   1:  PR[GP1:91,1] = PR[GP1:90,1] + -48.523;
   1:  PR[GP1:91,2] = PR[GP1:90,2] + 33.030;
   1:L PR[91] R[100]mm/sec CNT100;
   1:  PR[GP1:91,1] = PR[GP1:90,1] + -49.948;
   1:  PR[GP1:91,2] = PR[GP1:90,2] + 32.411;
   1:L PR[91] R[100]mm/sec CNT100;
   1:  PR[GP1:91,1] = PR[GP1:90,1] + -58.284;
   1:  PR[GP1:91,2] = PR[GP1:90,2] + 28.248;
   1:L PR[91] R[100]mm/sec CNT100;
   1:  PR[GP1:91,1] = PR[GP1:90,1] + -60.456;
   1:  PR[GP1:91,2] = PR[GP1:90,2] + 26.266;
   1:L PR[91] R[100]mm/sec CNT100;
   1:  PR[GP1:91,1] = PR[GP1:90,1] + -66.187;
   1:  PR[GP1:91,2] = PR[GP1:90,2] + 20.627;
   1:L PR[91] R[100]mm/sec CNT100;
   1:  PR[GP1:91,1] = PR[GP1:90,1] + -68.044;
   1:  PR[GP1:91,2] = PR[GP1:90,2] + 17.225;
   1:L PR[91] R[100]mm/sec CNT100;
   1:  PR[GP1:91,1] = PR[GP1:90,1] + -71.335;
   1:  PR[GP1:91,2] = PR[GP1:90,2] + 10.856;
   1:L PR[91] R[100]mm/sec CNT100;
   1:  PR[GP1:91,1] = PR[GP1:90,1] + -72.085;
   1:  PR[GP1:91,2] = PR[GP1:90,2] + 6.431;
   1:L PR[91] R[100]mm/sec CNT100;
   1:  PR[GP1:91,1] = PR[GP1:90,1] + -73.126;
   1:  PR[GP1:91,2] = PR[GP1:90,2] + -0.069;
   1:L PR[91] R[100]mm/sec CNT100;
   1:  PR[GP1:91,1] = PR[GP1:90,1] + -72.374;
   1:  PR[GP1:91,2] = PR[GP1:90,2] + -4.503;
   1:L PR[91] R[100]mm/sec CNT100;
   1:  PR[GP1:91,1] = PR[GP1:90,1] + -71.334;
   1:  PR[GP1:91,2] = PR[GP1:90,2] + -11.003;
   1:L PR[91] R[100]mm/sec CNT100;
   1:  PR[GP1:91,1] = PR[GP1:90,1] + -68.044;
   1:  PR[GP1:91,2] = PR[GP1:90,2] + -17.369;
   1:L PR[91] R[100]mm/sec CNT100;
   1:  PR[GP1:91,1] = PR[GP1:90,1] + -66.187;
   1:  PR[GP1:91,2] = PR[GP1:90,2] + -20.771;
   1:L PR[91] R[100]mm/sec CNT100;
   1:  PR[GP1:91,1] = PR[GP1:90,1] + -60.456;
   1:  PR[GP1:91,2] = PR[GP1:90,2] + -26.411;
   1:L PR[91] R[100]mm/sec CNT100;
   1:  PR[GP1:91,1] = PR[GP1:90,1] + -58.284;
   1:  PR[GP1:91,2] = PR[GP1:90,2] + -28.392;
   1:L PR[91] R[100]mm/sec CNT100;
   1:  PR[GP1:91,1] = PR[GP1:90,1] + -49.948;
   1:  PR[GP1:91,2] = PR[GP1:90,2] + -32.555;
   1:L PR[91] R[100]mm/sec CNT100;
   1:  PR[GP1:91,1] = PR[GP1:90,1] + -48.524;
   1:  PR[GP1:91,2] = PR[GP1:90,2] + -33.174;
   1:L PR[91] R[100]mm/sec CNT100;
   1:  PR[GP1:91,1] = PR[GP1:90,1] + -37.881;
   1:  PR[GP1:91,2] = PR[GP1:90,2] + -34.799;
   1:L PR[91] R[100]mm/sec CNT100;
   1:  PR[GP1:91,1] = PR[GP1:90,1] + -37.801;
   1:  PR[GP1:91,2] = PR[GP1:90,2] + -34.793;
   1:L PR[91] R[100]mm/sec CNT100;
   1:  PR[GP1:91,1] = PR[GP1:90,1] + -27.317;
   1:  PR[GP1:91,2] = PR[GP1:90,2] + -33.256;
   1:L PR[91] R[100]mm/sec CNT100;
   1:  PR[GP1:91,1] = PR[GP1:90,1] + -25.233;
   1:  PR[GP1:91,2] = PR[GP1:90,2] + -32.463;
   1:L PR[91] R[100]mm/sec CNT100;
   1:  PR[GP1:91,1] = PR[GP1:90,1] + -17.847;
   1:  PR[GP1:91,2] = PR[GP1:90,2] + -28.861;
   1:L PR[91] R[100]mm/sec CNT100;
   1:  PR[GP1:91,1] = PR[GP1:90,1] + -14.429;
   1:  PR[GP1:91,2] = PR[GP1:90,2] + -26.222;
   1:L PR[91] R[100]mm/sec CNT100;
   1:  PR[GP1:91,1] = PR[GP1:90,1] + -10.165;
   1:  PR[GP1:91,2] = PR[GP1:90,2] + -22.104;
   1:L PR[91] R[100]mm/sec CNT100;
   1:  PR[GP1:91,1] = PR[GP1:90,1] + -6.579;
   1:  PR[GP1:91,2] = PR[GP1:90,2] + -16.904;
   1:L PR[91] R[100]mm/sec CNT100;
   1:  PR[GP1:91,1] = PR[GP1:90,1] + -4.548;
   1:  PR[GP1:91,2] = PR[GP1:90,2] + -13.017;
   1:L PR[91] R[100]mm/sec CNT100;
   1:  PR[GP1:91,1] = PR[GP1:90,1] + -4.423;
   1:  PR[GP1:91,2] = PR[GP1:90,2] + -13.058;
   1:L PR[91] R[100]mm/sec CNT100;
   1:  PR[GP1:91,1] = PR[GP1:90,1] + -2.556;
   1:  PR[GP1:91,2] = PR[GP1:90,2] + -11.014;
   1:L PR[91] R[100]mm/sec CNT100;
   1:  PR[GP1:91,1] = PR[GP1:90,1] + -1.961;
   1:  PR[GP1:91,2] = PR[GP1:90,2] + -10.303;
   1:L PR[91] R[100]mm/sec CNT100;
   1:  PR[GP1:91,1] = PR[GP1:90,1] + -1.561;
   1:  PR[GP1:91,2] = PR[GP1:90,2] + -10.351;
   1:L PR[91] R[100]mm/sec CNT100;
   1:  PR[GP1:91,1] = PR[GP1:90,1] + 2.228;
   1:  PR[GP1:91,2] = PR[GP1:90,2] + -10.312;
   1:L PR[91] R[100]mm/sec CNT100;
   1:  PR[GP1:91,1] = PR[GP1:90,1] + 2.419;
   1:  PR[GP1:91,2] = PR[GP1:90,2] + -10.673;
   1:L PR[91] R[100]mm/sec CNT100;
   1:  PR[GP1:91,1] = PR[GP1:90,1] + 2.721;
   1:  PR[GP1:91,2] = PR[GP1:90,2] + -11.007;
   1:L PR[91] R[100]mm/sec CNT100;
   1:  PR[GP1:91,1] = PR[GP1:90,1] + 4.385;
   1:  PR[GP1:91,2] = PR[GP1:90,2] + -12.999;
   1:L PR[91] R[100]mm/sec CNT100;
   1:  PR[GP1:91,1] = PR[GP1:90,1] + 4.919;
   1:  PR[GP1:91,2] = PR[GP1:90,2] + -13.336;
   1:L PR[91] R[100]mm/sec CNT100;
   1:  PR[GP1:91,1] = PR[GP1:90,1] + 6.783;
   1:  PR[GP1:91,2] = PR[GP1:90,2] + -16.884;
   1:L PR[91] R[100]mm/sec CNT100;
   1:  PR[GP1:91,1] = PR[GP1:90,1] + 10.374;
   1:  PR[GP1:91,2] = PR[GP1:90,2] + -22.091;
   1:L PR[91] R[100]mm/sec CNT100;
   1:  PR[GP1:91,1] = PR[GP1:90,1] + 14.635;
   1:  PR[GP1:91,2] = PR[GP1:90,2] + -26.217;
   1:L PR[91] R[100]mm/sec CNT100;
   1:  PR[GP1:91,1] = PR[GP1:90,1] + 18.052;
   1:  PR[GP1:91,2] = PR[GP1:90,2] + -28.858;
   1:L PR[91] R[100]mm/sec CNT100;
   1:  PR[GP1:91,1] = PR[GP1:90,1] + 25.434;
   1:  PR[GP1:91,2] = PR[GP1:90,2] + -32.459;
   1:L PR[91] R[100]mm/sec CNT100;
   1:  PR[GP1:91,1] = PR[GP1:90,1] + 27.520;
   1:  PR[GP1:91,2] = PR[GP1:90,2] + -33.250;
   1:L PR[91] R[100]mm/sec CNT100;
   1:  PR[GP1:91,1] = PR[GP1:90,1] + 38.001;
   1:  PR[GP1:91,2] = PR[GP1:90,2] + -34.793;
   1:L PR[91] R[100]mm/sec CNT100;
   1:  PR[GP1:91,1] = PR[GP1:90,1] + 38.083;
   1:  PR[GP1:91,2] = PR[GP1:90,2] + -34.799;
   1:L PR[91] R[100]mm/sec CNT100;
   1:  PR[GP1:91,1] = PR[GP1:90,1] + 48.729;
   1:  PR[GP1:91,2] = PR[GP1:90,2] + -33.175;
   1:L PR[91] R[100]mm/sec CNT100;
   1:  PR[GP1:91,1] = PR[GP1:90,1] + 50.153;
   1:  PR[GP1:91,2] = PR[GP1:90,2] + -32.556;
   1:L PR[91] R[100]mm/sec CNT100;
   1:  PR[GP1:91,1] = PR[GP1:90,1] + 58.492;
   1:  PR[GP1:91,2] = PR[GP1:90,2] + -28.398;
   1:L PR[91] R[100]mm/sec CNT100;
   1:  PR[GP1:91,1] = PR[GP1:90,1] + 60.665;
   1:  PR[GP1:91,2] = PR[GP1:90,2] + -26.416;
   1:L PR[91] R[100]mm/sec CNT100;
   1:  PR[GP1:91,1] = PR[GP1:90,1] + 66.398;
   1:  PR[GP1:91,2] = PR[GP1:90,2] + -20.767;
   1:L PR[91] R[100]mm/sec CNT100;
   1:  PR[GP1:91,1] = PR[GP1:90,1] + 68.256;
   1:  PR[GP1:91,2] = PR[GP1:90,2] + -17.367;
   1:L PR[91] R[100]mm/sec CNT100;
   1:  PR[GP1:91,1] = PR[GP1:90,1] + 71.548;
   1:  PR[GP1:91,2] = PR[GP1:90,2] + -11.013;
   1:L PR[91] R[100]mm/sec CNT100;
   1:  PR[GP1:91,1] = PR[GP1:90,1] + 72.297;
   1:  PR[GP1:91,2] = PR[GP1:90,2] + -6.586;
   1:L PR[91] R[100]mm/sec CNT100;
   1:  PR[GP1:91,1] = PR[GP1:90,1] + 73.340;
   1:  PR[GP1:91,2] = PR[GP1:90,2] + -0.075;
   1:L PR[91] R[100]mm/sec CNT100;
   1:  PR[GP1:91,1] = PR[GP1:90,1] + 72.588;
   1:  PR[GP1:91,2] = PR[GP1:90,2] + 4.361;
   1:L PR[91] R[100]mm/sec CNT100;
   1:  PR[GP1:91,1] = PR[GP1:90,1] + 71.547;
   1:  PR[GP1:91,2] = PR[GP1:90,2] + 10.872;
   1:L PR[91] R[100]mm/sec CNT100;
   1:  PR[GP1:91,1] = PR[GP1:90,1] + 68.256;
   1:  PR[GP1:91,2] = PR[GP1:90,2] + 17.223;
   1:L PR[91] R[100]mm/sec CNT100;
   1:  PR[GP1:91,1] = PR[GP1:90,1] + 66.398;
   1:  PR[GP1:91,2] = PR[GP1:90,2] + 20.623;
   1:L PR[91] R[100]mm/sec CNT100;
   1:  PR[GP1:91,1] = PR[GP1:90,1] + 60.665;
   1:  PR[GP1:91,2] = PR[GP1:90,2] + 26.272;
   1:L PR[91] R[100]mm/sec CNT100;
   1:  PR[GP1:91,1] = PR[GP1:90,1] + 58.492;
   1:  PR[GP1:91,2] = PR[GP1:90,2] + 28.254;
   1:L PR[91] R[100]mm/sec CNT100;
   1:  PR[GP1:91,1] = PR[GP1:90,1] + 50.152;
   1:  PR[GP1:91,2] = PR[GP1:90,2] + 32.412;
   1:L PR[91] R[100]mm/sec CNT100;
   1:  PR[GP1:91,1] = PR[GP1:90,1] + 48.729;
   1:  PR[GP1:91,2] = PR[GP1:90,2] + 33.031;
   1:L PR[91] R[100]mm/sec CNT100;
   1:  PR[GP1:91,1] = PR[GP1:90,1] + 38.083;
   1:  PR[GP1:91,2] = PR[GP1:90,2] + 34.655;
   1:L PR[91] R[100]mm/sec CNT100;
   1:  PR[GP1:91,1] = PR[GP1:90,1] + 38.001;
   1:  PR[GP1:91,2] = PR[GP1:90,2] + 34.649;
   1:L PR[91] R[100]mm/sec CNT100;
   1:  PR[GP1:91,1] = PR[GP1:90,1] + 27.520;
   1:  PR[GP1:91,2] = PR[GP1:90,2] + 33.106;
   1:L PR[91] R[100]mm/sec CNT100;
   1:  PR[GP1:91,1] = PR[GP1:90,1] + 25.434;
   1:  PR[GP1:91,2] = PR[GP1:90,2] + 32.314;
   1:L PR[91] R[100]mm/sec CNT100;
   1:  PR[GP1:91,1] = PR[GP1:90,1] + 18.052;
   1:  PR[GP1:91,2] = PR[GP1:90,2] + 28.714;
   1:L PR[91] R[100]mm/sec CNT100;
   1:  PR[GP1:91,1] = PR[GP1:90,1] + 14.635;
   1:  PR[GP1:91,2] = PR[GP1:90,2] + 26.073;
   1:L PR[91] R[100]mm/sec CNT100;
   1:  PR[GP1:91,1] = PR[GP1:90,1] + 10.374;
   1:  PR[GP1:91,2] = PR[GP1:90,2] + 21.947;
   1:L PR[91] R[100]mm/sec CNT100;
   1:  PR[GP1:91,1] = PR[GP1:90,1] + 6.797;
   1:  PR[GP1:91,2] = PR[GP1:90,2] + 16.767;
   1:L PR[91] R[100]mm/sec CNT100;
   1:  PR[GP1:91,1] = PR[GP1:90,1] + 4.956;
   1:  PR[GP1:91,2] = PR[GP1:90,2] + 13.264;
   1:L PR[91] R[100]mm/sec CNT100;
   1:  PR[GP1:91,1] = PR[GP1:90,1] + 2.737;
   1:  PR[GP1:91,2] = PR[GP1:90,2] + 10.879;
   1:L PR[91] R[100]mm/sec CNT100;
   1:  PR[GP1:91,1] = PR[GP1:90,1] + 2.140;
   1:  PR[GP1:91,2] = PR[GP1:90,2] + 10.164;
   1:L PR[91] R[100]mm/sec CNT100;
   1:  PR[GP1:91,1] = PR[GP1:90,1] + -1.651;
   1:  PR[GP1:91,2] = PR[GP1:90,2] + 10.194;
   1:L PR[91] R[100]mm/sec CNT100;
   1:  ! -- Layer/Ebene 45 -- !;
   1:  PR[91] = PR[90];
   1:  PR[GP1:91,1] = PR[GP1:90,1] + -2.160;
   1:  PR[GP1:91,2] = PR[GP1:90,2] + 10.865;
   1:  PR[GP1:91,3] = PR[GP1:90,3] + 27.755;
   1:L PR[91] R[100]mm/sec CNT100;
   1:  PR[GP1:91,1] = PR[GP1:90,1] + -4.791;
   1:  PR[GP1:91,2] = PR[GP1:90,2] + 13.704;
   1:L PR[91] R[100]mm/sec CNT100;
   1:  PR[GP1:91,1] = PR[GP1:90,1] + -4.807;
   1:  PR[GP1:91,2] = PR[GP1:90,2] + 13.843;
   1:L PR[91] R[100]mm/sec CNT100;
   1:  PR[GP1:91,1] = PR[GP1:90,1] + -6.082;
   1:  PR[GP1:91,2] = PR[GP1:90,2] + 16.274;
   1:L PR[91] R[100]mm/sec CNT100;
   1:  PR[GP1:91,1] = PR[GP1:90,1] + -10.209;
   1:  PR[GP1:91,2] = PR[GP1:90,2] + 22.252;
   1:L PR[91] R[100]mm/sec CNT100;
   1:  PR[GP1:91,1] = PR[GP1:90,1] + -13.777;
   1:  PR[GP1:91,2] = PR[GP1:90,2] + 25.698;
   1:L PR[91] R[100]mm/sec CNT100;
   1:  PR[GP1:91,1] = PR[GP1:90,1] + -17.920;
   1:  PR[GP1:91,2] = PR[GP1:90,2] + 28.896;
   1:L PR[91] R[100]mm/sec CNT100;
   1:  PR[GP1:91,1] = PR[GP1:90,1] + -24.472;
   1:  PR[GP1:91,2] = PR[GP1:90,2] + 32.093;
   1:L PR[91] R[100]mm/sec CNT100;
   1:  PR[GP1:91,1] = PR[GP1:90,1] + -27.383;
   1:  PR[GP1:91,2] = PR[GP1:90,2] + 33.199;
   1:L PR[91] R[100]mm/sec CNT100;
   1:  PR[GP1:91,1] = PR[GP1:90,1] + -37.001;
   1:  PR[GP1:91,2] = PR[GP1:90,2] + 34.610;
   1:L PR[91] R[100]mm/sec CNT100;
   1:  PR[GP1:91,1] = PR[GP1:90,1] + -37.913;
   1:  PR[GP1:91,2] = PR[GP1:90,2] + 34.674;
   1:L PR[91] R[100]mm/sec CNT100;
   1:  PR[GP1:91,1] = PR[GP1:90,1] + -43.210;
   1:  PR[GP1:91,2] = PR[GP1:90,2] + 33.821;
   1:L PR[91] R[100]mm/sec CNT100;
   1:  PR[GP1:91,1] = PR[GP1:90,1] + -48.579;
   1:  PR[GP1:91,2] = PR[GP1:90,2] + 33.005;
   1:L PR[91] R[100]mm/sec CNT100;
   1:  PR[GP1:91,1] = PR[GP1:90,1] + -49.324;
   1:  PR[GP1:91,2] = PR[GP1:90,2] + 32.681;
   1:L PR[91] R[100]mm/sec CNT100;
   1:  PR[GP1:91,1] = PR[GP1:90,1] + -58.292;
   1:  PR[GP1:91,2] = PR[GP1:90,2] + 28.203;
   1:L PR[91] R[100]mm/sec CNT100;
   1:  PR[GP1:91,1] = PR[GP1:90,1] + -59.957;
   1:  PR[GP1:91,2] = PR[GP1:90,2] + 26.684;
   1:L PR[91] R[100]mm/sec CNT100;
   1:  PR[GP1:91,1] = PR[GP1:90,1] + -66.156;
   1:  PR[GP1:91,2] = PR[GP1:90,2] + 20.584;
   1:L PR[91] R[100]mm/sec CNT100;
   1:  PR[GP1:91,1] = PR[GP1:90,1] + -67.704;
   1:  PR[GP1:91,2] = PR[GP1:90,2] + 17.748;
   1:L PR[91] R[100]mm/sec CNT100;
   1:  PR[GP1:91,1] = PR[GP1:90,1] + -71.279;
   1:  PR[GP1:91,2] = PR[GP1:90,2] + 10.831;
   1:L PR[91] R[100]mm/sec CNT100;
   1:  PR[GP1:91,1] = PR[GP1:90,1] + -71.922;
   1:  PR[GP1:91,2] = PR[GP1:90,2] + 7.028;
   1:L PR[91] R[100]mm/sec CNT100;
   1:  PR[GP1:91,1] = PR[GP1:90,1] + -73.060;
   1:  PR[GP1:91,2] = PR[GP1:90,2] + -0.069;
   1:L PR[91] R[100]mm/sec CNT100;
   1:  PR[GP1:91,1] = PR[GP1:90,1] + -72.407;
   1:  PR[GP1:91,2] = PR[GP1:90,2] + -3.918;
   1:L PR[91] R[100]mm/sec CNT100;
   1:  PR[GP1:91,1] = PR[GP1:90,1] + -71.277;
   1:  PR[GP1:91,2] = PR[GP1:90,2] + -10.977;
   1:L PR[91] R[100]mm/sec CNT100;
   1:  PR[GP1:91,1] = PR[GP1:90,1] + -67.704;
   1:  PR[GP1:91,2] = PR[GP1:90,2] + -17.892;
   1:L PR[91] R[100]mm/sec CNT100;
   1:  PR[GP1:91,1] = PR[GP1:90,1] + -66.156;
   1:  PR[GP1:91,2] = PR[GP1:90,2] + -20.728;
   1:L PR[91] R[100]mm/sec CNT100;
   1:  PR[GP1:91,1] = PR[GP1:90,1] + -59.957;
   1:  PR[GP1:91,2] = PR[GP1:90,2] + -26.828;
   1:L PR[91] R[100]mm/sec CNT100;
   1:  PR[GP1:91,1] = PR[GP1:90,1] + -58.292;
   1:  PR[GP1:91,2] = PR[GP1:90,2] + -28.347;
   1:L PR[91] R[100]mm/sec CNT100;
   1:  PR[GP1:91,1] = PR[GP1:90,1] + -49.325;
   1:  PR[GP1:91,2] = PR[GP1:90,2] + -32.825;
   1:L PR[91] R[100]mm/sec CNT100;
   1:  PR[GP1:91,1] = PR[GP1:90,1] + -48.579;
   1:  PR[GP1:91,2] = PR[GP1:90,2] + -33.149;
   1:L PR[91] R[100]mm/sec CNT100;
   1:  PR[GP1:91,1] = PR[GP1:90,1] + -43.210;
   1:  PR[GP1:91,2] = PR[GP1:90,2] + -33.965;
   1:L PR[91] R[100]mm/sec CNT100;
   1:  PR[GP1:91,1] = PR[GP1:90,1] + -37.913;
   1:  PR[GP1:91,2] = PR[GP1:90,2] + -34.818;
   1:L PR[91] R[100]mm/sec CNT100;
   1:  PR[GP1:91,1] = PR[GP1:90,1] + -37.002;
   1:  PR[GP1:91,2] = PR[GP1:90,2] + -34.754;
   1:L PR[91] R[100]mm/sec CNT100;
   1:  PR[GP1:91,1] = PR[GP1:90,1] + -27.383;
   1:  PR[GP1:91,2] = PR[GP1:90,2] + -33.343;
   1:L PR[91] R[100]mm/sec CNT100;
   1:  PR[GP1:91,1] = PR[GP1:90,1] + -24.472;
   1:  PR[GP1:91,2] = PR[GP1:90,2] + -32.237;
   1:L PR[91] R[100]mm/sec CNT100;
   1:  PR[GP1:91,1] = PR[GP1:90,1] + -17.920;
   1:  PR[GP1:91,2] = PR[GP1:90,2] + -29.041;
   1:L PR[91] R[100]mm/sec CNT100;
   1:  PR[GP1:91,1] = PR[GP1:90,1] + -13.777;
   1:  PR[GP1:91,2] = PR[GP1:90,2] + -25.842;
   1:L PR[91] R[100]mm/sec CNT100;
   1:  PR[GP1:91,1] = PR[GP1:90,1] + -10.210;
   1:  PR[GP1:91,2] = PR[GP1:90,2] + -22.396;
   1:L PR[91] R[100]mm/sec CNT100;
   1:  PR[GP1:91,1] = PR[GP1:90,1] + -6.066;
   1:  PR[GP1:91,2] = PR[GP1:90,2] + -16.388;
   1:L PR[91] R[100]mm/sec CNT100;
   1:  PR[GP1:91,1] = PR[GP1:90,1] + -4.516;
   1:  PR[GP1:91,2] = PR[GP1:90,2] + -13.422;
   1:L PR[91] R[100]mm/sec CNT100;
   1:  PR[GP1:91,1] = PR[GP1:90,1] + -4.394;
   1:  PR[GP1:91,2] = PR[GP1:90,2] + -13.462;
   1:L PR[91] R[100]mm/sec CNT100;
   1:  PR[GP1:91,1] = PR[GP1:90,1] + -2.162;
   1:  PR[GP1:91,2] = PR[GP1:90,2] + -11.011;
   1:L PR[91] R[100]mm/sec CNT100;
   1:  PR[GP1:91,1] = PR[GP1:90,1] + -1.823;
   1:  PR[GP1:91,2] = PR[GP1:90,2] + -10.812;
   1:L PR[91] R[100]mm/sec CNT100;
   1:  PR[GP1:91,1] = PR[GP1:90,1] + 2.075;
   1:  PR[GP1:91,2] = PR[GP1:90,2] + -10.774;
   1:L PR[91] R[100]mm/sec CNT100;
   1:  PR[GP1:91,1] = PR[GP1:90,1] + 4.171;
   1:  PR[GP1:91,2] = PR[GP1:90,2] + -13.284;
   1:L PR[91] R[100]mm/sec CNT100;
   1:  PR[GP1:91,1] = PR[GP1:90,1] + 4.886;
   1:  PR[GP1:91,2] = PR[GP1:90,2] + -13.736;
   1:L PR[91] R[100]mm/sec CNT100;
   1:  PR[GP1:91,1] = PR[GP1:90,1] + 6.270;
   1:  PR[GP1:91,2] = PR[GP1:90,2] + -16.369;
   1:L PR[91] R[100]mm/sec CNT100;
   1:  PR[GP1:91,1] = PR[GP1:90,1] + 10.419;
   1:  PR[GP1:91,2] = PR[GP1:90,2] + -22.385;
   1:L PR[91] R[100]mm/sec CNT100;
   1:  PR[GP1:91,1] = PR[GP1:90,1] + 13.984;
   1:  PR[GP1:91,2] = PR[GP1:90,2] + -25.837;
   1:L PR[91] R[100]mm/sec CNT100;
   1:  PR[GP1:91,1] = PR[GP1:90,1] + 18.126;
   1:  PR[GP1:91,2] = PR[GP1:90,2] + -29.039;
   1:L PR[91] R[100]mm/sec CNT100;
   1:  PR[GP1:91,1] = PR[GP1:90,1] + 24.675;
   1:  PR[GP1:91,2] = PR[GP1:90,2] + -32.233;
   1:L PR[91] R[100]mm/sec CNT100;
   1:  PR[GP1:91,1] = PR[GP1:90,1] + 27.587;
   1:  PR[GP1:91,2] = PR[GP1:90,2] + -33.338;
   1:L PR[91] R[100]mm/sec CNT100;
   1:  PR[GP1:91,1] = PR[GP1:90,1] + 37.203;
   1:  PR[GP1:91,2] = PR[GP1:90,2] + -34.754;
   1:L PR[91] R[100]mm/sec CNT100;
   1:  PR[GP1:91,1] = PR[GP1:90,1] + 38.116;
   1:  PR[GP1:91,2] = PR[GP1:90,2] + -34.819;
   1:L PR[91] R[100]mm/sec CNT100;
   1:  PR[GP1:91,1] = PR[GP1:90,1] + 43.423;
   1:  PR[GP1:91,2] = PR[GP1:90,2] + -33.964;
   1:L PR[91] R[100]mm/sec CNT100;
   1:  PR[GP1:91,1] = PR[GP1:90,1] + 48.784;
   1:  PR[GP1:91,2] = PR[GP1:90,2] + -33.150;
   1:L PR[91] R[100]mm/sec CNT100;
   1:  PR[GP1:91,1] = PR[GP1:90,1] + 49.528;
   1:  PR[GP1:91,2] = PR[GP1:90,2] + -32.826;
   1:L PR[91] R[100]mm/sec CNT100;
   1:  PR[GP1:91,1] = PR[GP1:90,1] + 58.500;
   1:  PR[GP1:91,2] = PR[GP1:90,2] + -28.353;
   1:L PR[91] R[100]mm/sec CNT100;
   1:  PR[GP1:91,1] = PR[GP1:90,1] + 60.165;
   1:  PR[GP1:91,2] = PR[GP1:90,2] + -26.835;
   1:L PR[91] R[100]mm/sec CNT100;
   1:  PR[GP1:91,1] = PR[GP1:90,1] + 66.367;
   1:  PR[GP1:91,2] = PR[GP1:90,2] + -20.723;
   1:L PR[91] R[100]mm/sec CNT100;
   1:  PR[GP1:91,1] = PR[GP1:90,1] + 67.915;
   1:  PR[GP1:91,2] = PR[GP1:90,2] + -17.889;
   1:L PR[91] R[100]mm/sec CNT100;
   1:  PR[GP1:91,1] = PR[GP1:90,1] + 71.491;
   1:  PR[GP1:91,2] = PR[GP1:90,2] + -10.988;
   1:L PR[91] R[100]mm/sec CNT100;
   1:  PR[GP1:91,1] = PR[GP1:90,1] + 72.135;
   1:  PR[GP1:91,2] = PR[GP1:90,2] + -7.183;
   1:L PR[91] R[100]mm/sec CNT100;
   1:  PR[GP1:91,1] = PR[GP1:90,1] + 73.273;
   1:  PR[GP1:91,2] = PR[GP1:90,2] + -0.075;
   1:L PR[91] R[100]mm/sec CNT100;
   1:  PR[GP1:91,1] = PR[GP1:90,1] + 72.620;
   1:  PR[GP1:91,2] = PR[GP1:90,2] + 3.775;
   1:L PR[91] R[100]mm/sec CNT100;
   1:  PR[GP1:91,1] = PR[GP1:90,1] + 71.490;
   1:  PR[GP1:91,2] = PR[GP1:90,2] + 10.847;
   1:L PR[91] R[100]mm/sec CNT100;
   1:  PR[GP1:91,1] = PR[GP1:90,1] + 67.915;
   1:  PR[GP1:91,2] = PR[GP1:90,2] + 17.745;
   1:L PR[91] R[100]mm/sec CNT100;
   1:  PR[GP1:91,1] = PR[GP1:90,1] + 66.367;
   1:  PR[GP1:91,2] = PR[GP1:90,2] + 20.579;
   1:L PR[91] R[100]mm/sec CNT100;
   1:  PR[GP1:91,1] = PR[GP1:90,1] + 60.165;
   1:  PR[GP1:91,2] = PR[GP1:90,2] + 26.691;
   1:L PR[91] R[100]mm/sec CNT100;
   1:  PR[GP1:91,1] = PR[GP1:90,1] + 58.500;
   1:  PR[GP1:91,2] = PR[GP1:90,2] + 28.209;
   1:L PR[91] R[100]mm/sec CNT100;
   1:  PR[GP1:91,1] = PR[GP1:90,1] + 49.528;
   1:  PR[GP1:91,2] = PR[GP1:90,2] + 32.682;
   1:L PR[91] R[100]mm/sec CNT100;
   1:  PR[GP1:91,1] = PR[GP1:90,1] + 48.784;
   1:  PR[GP1:91,2] = PR[GP1:90,2] + 33.006;
   1:L PR[91] R[100]mm/sec CNT100;
   1:  PR[GP1:91,1] = PR[GP1:90,1] + 43.423;
   1:  PR[GP1:91,2] = PR[GP1:90,2] + 33.820;
   1:L PR[91] R[100]mm/sec CNT100;
   1:  PR[GP1:91,1] = PR[GP1:90,1] + 38.116;
   1:  PR[GP1:91,2] = PR[GP1:90,2] + 34.675;
   1:L PR[91] R[100]mm/sec CNT100;
   1:  PR[GP1:91,1] = PR[GP1:90,1] + 37.203;
   1:  PR[GP1:91,2] = PR[GP1:90,2] + 34.610;
   1:L PR[91] R[100]mm/sec CNT100;
   1:  PR[GP1:91,1] = PR[GP1:90,1] + 27.586;
   1:  PR[GP1:91,2] = PR[GP1:90,2] + 33.194;
   1:L PR[91] R[100]mm/sec CNT100;
   1:  PR[GP1:91,1] = PR[GP1:90,1] + 24.675;
   1:  PR[GP1:91,2] = PR[GP1:90,2] + 32.089;
   1:L PR[91] R[100]mm/sec CNT100;
   1:  PR[GP1:91,1] = PR[GP1:90,1] + 18.126;
   1:  PR[GP1:91,2] = PR[GP1:90,2] + 28.895;
   1:L PR[91] R[100]mm/sec CNT100;
   1:  PR[GP1:91,1] = PR[GP1:90,1] + 13.984;
   1:  PR[GP1:91,2] = PR[GP1:90,2] + 25.693;
   1:L PR[91] R[100]mm/sec CNT100;
   1:  PR[GP1:91,1] = PR[GP1:90,1] + 10.419;
   1:  PR[GP1:91,2] = PR[GP1:90,2] + 22.241;
   1:L PR[91] R[100]mm/sec CNT100;
   1:  PR[GP1:91,1] = PR[GP1:90,1] + 6.286;
   1:  PR[GP1:91,2] = PR[GP1:90,2] + 16.256;
   1:L PR[91] R[100]mm/sec CNT100;
   1:  PR[GP1:91,1] = PR[GP1:90,1] + 4.924;
   1:  PR[GP1:91,2] = PR[GP1:90,2] + 13.664;
   1:L PR[91] R[100]mm/sec CNT100;
   1:  PR[GP1:91,1] = PR[GP1:90,1] + 2.293;
   1:  PR[GP1:91,2] = PR[GP1:90,2] + 10.828;
   1:L PR[91] R[100]mm/sec CNT100;
   1:  PR[GP1:91,1] = PR[GP1:90,1] + 1.956;
   1:  PR[GP1:91,2] = PR[GP1:90,2] + 10.631;
   1:L PR[91] R[100]mm/sec CNT100;
   1:  PR[GP1:91,1] = PR[GP1:90,1] + -1.823;
   1:  PR[GP1:91,2] = PR[GP1:90,2] + 10.668;
   1:L PR[91] R[100]mm/sec CNT100;
   1:  ! -- Layer/Ebene 46 -- !;
   1:  PR[91] = PR[90];
   1:  PR[GP1:91,1] = PR[GP1:90,1] + -2.283;
   1:  PR[GP1:91,2] = PR[GP1:90,2] + 11.419;
   1:  PR[GP1:91,3] = PR[GP1:90,3] + 28.365;
   1:L PR[91] R[100]mm/sec CNT100;
   1:  PR[GP1:91,1] = PR[GP1:90,1] + -4.757;
   1:  PR[GP1:91,2] = PR[GP1:90,2] + 14.088;
   1:L PR[91] R[100]mm/sec CNT100;
   1:  PR[GP1:91,1] = PR[GP1:90,1] + -4.774;
   1:  PR[GP1:91,2] = PR[GP1:90,2] + 14.244;
   1:L PR[91] R[100]mm/sec CNT100;
   1:  PR[GP1:91,1] = PR[GP1:90,1] + -5.571;
   1:  PR[GP1:91,2] = PR[GP1:90,2] + 15.762;
   1:L PR[91] R[100]mm/sec CNT100;
   1:  PR[GP1:91,1] = PR[GP1:90,1] + -10.253;
   1:  PR[GP1:91,2] = PR[GP1:90,2] + 22.545;
   1:L PR[91] R[100]mm/sec CNT100;
   1:  PR[GP1:91,1] = PR[GP1:90,1] + -13.124;
   1:  PR[GP1:91,2] = PR[GP1:90,2] + 25.317;
   1:L PR[91] R[100]mm/sec CNT100;
   1:  PR[GP1:91,1] = PR[GP1:90,1] + -17.993;
   1:  PR[GP1:91,2] = PR[GP1:90,2] + 29.076;
   1:L PR[91] R[100]mm/sec CNT100;
   1:  PR[GP1:91,1] = PR[GP1:90,1] + -23.712;
   1:  PR[GP1:91,2] = PR[GP1:90,2] + 31.866;
   1:L PR[91] R[100]mm/sec CNT100;
   1:  PR[GP1:91,1] = PR[GP1:90,1] + -27.448;
   1:  PR[GP1:91,2] = PR[GP1:90,2] + 33.286;
   1:L PR[91] R[100]mm/sec CNT100;
   1:  PR[GP1:91,1] = PR[GP1:90,1] + -36.202;
   1:  PR[GP1:91,2] = PR[GP1:90,2] + 34.570;
   1:L PR[91] R[100]mm/sec CNT100;
   1:  PR[GP1:91,1] = PR[GP1:90,1] + -37.947;
   1:  PR[GP1:91,2] = PR[GP1:90,2] + 34.694;
   1:L PR[91] R[100]mm/sec CNT100;
   1:  PR[GP1:91,1] = PR[GP1:90,1] + -48.615;
   1:  PR[GP1:91,2] = PR[GP1:90,2] + 32.984;
   1:L PR[91] R[100]mm/sec CNT100;
   1:  PR[GP1:91,1] = PR[GP1:90,1] + -58.300;
   1:  PR[GP1:91,2] = PR[GP1:90,2] + 28.157;
   1:L PR[91] R[100]mm/sec CNT100;
   1:  PR[GP1:91,1] = PR[GP1:90,1] + -59.458;
   1:  PR[GP1:91,2] = PR[GP1:90,2] + 27.102;
   1:L PR[91] R[100]mm/sec CNT100;
   1:  PR[GP1:91,1] = PR[GP1:90,1] + -66.125;
   1:  PR[GP1:91,2] = PR[GP1:90,2] + 20.540;
   1:L PR[91] R[100]mm/sec CNT100;
   1:  PR[GP1:91,1] = PR[GP1:90,1] + -67.364;
   1:  PR[GP1:91,2] = PR[GP1:90,2] + 18.271;
   1:L PR[91] R[100]mm/sec CNT100;
   1:  PR[GP1:91,1] = PR[GP1:90,1] + -71.222;
   1:  PR[GP1:91,2] = PR[GP1:90,2] + 10.806;
   1:L PR[91] R[100]mm/sec CNT100;
   1:  PR[GP1:91,1] = PR[GP1:90,1] + -71.760;
   1:  PR[GP1:91,2] = PR[GP1:90,2] + 7.624;
   1:L PR[91] R[100]mm/sec CNT100;
   1:  PR[GP1:91,1] = PR[GP1:90,1] + -72.993;
   1:  PR[GP1:91,2] = PR[GP1:90,2] + -0.069;
   1:L PR[91] R[100]mm/sec CNT100;
   1:  PR[GP1:91,1] = PR[GP1:90,1] + -72.440;
   1:  PR[GP1:91,2] = PR[GP1:90,2] + -3.332;
   1:L PR[91] R[100]mm/sec CNT100;
   1:  PR[GP1:91,1] = PR[GP1:90,1] + -71.221;
   1:  PR[GP1:91,2] = PR[GP1:90,2] + -10.952;
   1:L PR[91] R[100]mm/sec CNT100;
   1:  PR[GP1:91,1] = PR[GP1:90,1] + -67.364;
   1:  PR[GP1:91,2] = PR[GP1:90,2] + -18.415;
   1:L PR[91] R[100]mm/sec CNT100;
   1:  PR[GP1:91,1] = PR[GP1:90,1] + -66.125;
   1:  PR[GP1:91,2] = PR[GP1:90,2] + -20.684;
   1:L PR[91] R[100]mm/sec CNT100;
   1:  PR[GP1:91,1] = PR[GP1:90,1] + -59.458;
   1:  PR[GP1:91,2] = PR[GP1:90,2] + -27.246;
   1:L PR[91] R[100]mm/sec CNT100;
   1:  PR[GP1:91,1] = PR[GP1:90,1] + -58.300;
   1:  PR[GP1:91,2] = PR[GP1:90,2] + -28.301;
   1:L PR[91] R[100]mm/sec CNT100;
   1:  PR[GP1:91,1] = PR[GP1:90,1] + -48.615;
   1:  PR[GP1:91,2] = PR[GP1:90,2] + -33.128;
   1:L PR[91] R[100]mm/sec CNT100;
   1:  PR[GP1:91,1] = PR[GP1:90,1] + -37.947;
   1:  PR[GP1:91,2] = PR[GP1:90,2] + -34.838;
   1:L PR[91] R[100]mm/sec CNT100;
   1:  PR[GP1:91,1] = PR[GP1:90,1] + -36.202;
   1:  PR[GP1:91,2] = PR[GP1:90,2] + -34.714;
   1:L PR[91] R[100]mm/sec CNT100;
   1:  PR[GP1:91,1] = PR[GP1:90,1] + -27.448;
   1:  PR[GP1:91,2] = PR[GP1:90,2] + -33.430;
   1:L PR[91] R[100]mm/sec CNT100;
   1:  PR[GP1:91,1] = PR[GP1:90,1] + -23.712;
   1:  PR[GP1:91,2] = PR[GP1:90,2] + -32.010;
   1:L PR[91] R[100]mm/sec CNT100;
   1:  PR[GP1:91,1] = PR[GP1:90,1] + -17.993;
   1:  PR[GP1:91,2] = PR[GP1:90,2] + -29.220;
   1:L PR[91] R[100]mm/sec CNT100;
   1:  PR[GP1:91,1] = PR[GP1:90,1] + -13.124;
   1:  PR[GP1:91,2] = PR[GP1:90,2] + -25.461;
   1:L PR[91] R[100]mm/sec CNT100;
   1:  PR[GP1:91,1] = PR[GP1:90,1] + -10.254;
   1:  PR[GP1:91,2] = PR[GP1:90,2] + -22.689;
   1:L PR[91] R[100]mm/sec CNT100;
   1:  PR[GP1:91,1] = PR[GP1:90,1] + -5.552;
   1:  PR[GP1:91,2] = PR[GP1:90,2] + -15.872;
   1:L PR[91] R[100]mm/sec CNT100;
   1:  PR[GP1:91,1] = PR[GP1:90,1] + -4.684;
   1:  PR[GP1:91,2] = PR[GP1:90,2] + -14.210;
   1:L PR[91] R[100]mm/sec CNT100;
   1:  PR[GP1:91,1] = PR[GP1:90,1] + -3.287;
   1:  PR[GP1:91,2] = PR[GP1:90,2] + -12.688;
   1:L PR[91] R[100]mm/sec CNT100;
   1:  PR[GP1:91,1] = PR[GP1:90,1] + -2.288;
   1:  PR[GP1:91,2] = PR[GP1:90,2] + -11.566;
   1:L PR[91] R[100]mm/sec CNT100;
   1:  PR[GP1:91,1] = PR[GP1:90,1] + -1.719;
   1:  PR[GP1:91,2] = PR[GP1:90,2] + -11.234;
   1:L PR[91] R[100]mm/sec CNT100;
   1:  PR[GP1:91,1] = PR[GP1:90,1] + 1.976;
   1:  PR[GP1:91,2] = PR[GP1:90,2] + -11.198;
   1:L PR[91] R[100]mm/sec CNT100;
   1:  PR[GP1:91,1] = PR[GP1:90,1] + 3.956;
   1:  PR[GP1:91,2] = PR[GP1:90,2] + -13.570;
   1:L PR[91] R[100]mm/sec CNT100;
   1:  PR[GP1:91,1] = PR[GP1:90,1] + 4.854;
   1:  PR[GP1:91,2] = PR[GP1:90,2] + -14.136;
   1:L PR[91] R[100]mm/sec CNT100;
   1:  PR[GP1:91,1] = PR[GP1:90,1] + 5.757;
   1:  PR[GP1:91,2] = PR[GP1:90,2] + -15.854;
   1:L PR[91] R[100]mm/sec CNT100;
   1:  PR[GP1:91,1] = PR[GP1:90,1] + 10.464;
   1:  PR[GP1:91,2] = PR[GP1:90,2] + -22.679;
   1:L PR[91] R[100]mm/sec CNT100;
   1:  PR[GP1:91,1] = PR[GP1:90,1] + 13.332;
   1:  PR[GP1:91,2] = PR[GP1:90,2] + -25.457;
   1:L PR[91] R[100]mm/sec CNT100;
   1:  PR[GP1:91,1] = PR[GP1:90,1] + 18.200;
   1:  PR[GP1:91,2] = PR[GP1:90,2] + -29.220;
   1:L PR[91] R[100]mm/sec CNT100;
   1:  PR[GP1:91,1] = PR[GP1:90,1] + 23.916;
   1:  PR[GP1:91,2] = PR[GP1:90,2] + -32.007;
   1:L PR[91] R[100]mm/sec CNT100;
   1:  PR[GP1:91,1] = PR[GP1:90,1] + 27.653;
   1:  PR[GP1:91,2] = PR[GP1:90,2] + -33.425;
   1:L PR[91] R[100]mm/sec CNT100;
   1:  PR[GP1:91,1] = PR[GP1:90,1] + 36.404;
   1:  PR[GP1:91,2] = PR[GP1:90,2] + -34.714;
   1:L PR[91] R[100]mm/sec CNT100;
   1:  PR[GP1:91,1] = PR[GP1:90,1] + 38.151;
   1:  PR[GP1:91,2] = PR[GP1:90,2] + -34.838;
   1:L PR[91] R[100]mm/sec CNT100;
   1:  PR[GP1:91,1] = PR[GP1:90,1] + 48.820;
   1:  PR[GP1:91,2] = PR[GP1:90,2] + -33.129;
   1:L PR[91] R[100]mm/sec CNT100;
   1:  PR[GP1:91,1] = PR[GP1:90,1] + 58.509;
   1:  PR[GP1:91,2] = PR[GP1:90,2] + -28.308;
   1:L PR[91] R[100]mm/sec CNT100;
   1:  PR[GP1:91,1] = PR[GP1:90,1] + 59.665;
   1:  PR[GP1:91,2] = PR[GP1:90,2] + -27.253;
   1:L PR[91] R[100]mm/sec CNT100;
   1:  PR[GP1:91,1] = PR[GP1:90,1] + 66.336;
   1:  PR[GP1:91,2] = PR[GP1:90,2] + -20.680;
   1:L PR[91] R[100]mm/sec CNT100;
   1:  PR[GP1:91,1] = PR[GP1:90,1] + 67.575;
   1:  PR[GP1:91,2] = PR[GP1:90,2] + -18.412;
   1:L PR[91] R[100]mm/sec CNT100;
   1:  PR[GP1:91,1] = PR[GP1:90,1] + 71.435;
   1:  PR[GP1:91,2] = PR[GP1:90,2] + -10.964;
   1:L PR[91] R[100]mm/sec CNT100;
   1:  PR[GP1:91,1] = PR[GP1:90,1] + 71.973;
   1:  PR[GP1:91,2] = PR[GP1:90,2] + -7.781;
   1:L PR[91] R[100]mm/sec CNT100;
   1:  PR[GP1:91,1] = PR[GP1:90,1] + 73.207;
   1:  PR[GP1:91,2] = PR[GP1:90,2] + -0.075;
   1:L PR[91] R[100]mm/sec CNT100;
   1:  PR[GP1:91,1] = PR[GP1:90,1] + 72.653;
   1:  PR[GP1:91,2] = PR[GP1:90,2] + 3.190;
   1:L PR[91] R[100]mm/sec CNT100;
   1:  PR[GP1:91,1] = PR[GP1:90,1] + 71.433;
   1:  PR[GP1:91,2] = PR[GP1:90,2] + 10.822;
   1:L PR[91] R[100]mm/sec CNT100;
   1:  PR[GP1:91,1] = PR[GP1:90,1] + 67.575;
   1:  PR[GP1:91,2] = PR[GP1:90,2] + 18.268;
   1:L PR[91] R[100]mm/sec CNT100;
   1:  PR[GP1:91,1] = PR[GP1:90,1] + 66.336;
   1:  PR[GP1:91,2] = PR[GP1:90,2] + 20.536;
   1:L PR[91] R[100]mm/sec CNT100;
   1:  PR[GP1:91,1] = PR[GP1:90,1] + 59.665;
   1:  PR[GP1:91,2] = PR[GP1:90,2] + 27.109;
   1:L PR[91] R[100]mm/sec CNT100;
   1:  PR[GP1:91,1] = PR[GP1:90,1] + 58.509;
   1:  PR[GP1:91,2] = PR[GP1:90,2] + 28.164;
   1:L PR[91] R[100]mm/sec CNT100;
   1:  PR[GP1:91,1] = PR[GP1:90,1] + 48.820;
   1:  PR[GP1:91,2] = PR[GP1:90,2] + 32.985;
   1:L PR[91] R[100]mm/sec CNT100;
   1:  PR[GP1:91,1] = PR[GP1:90,1] + 38.151;
   1:  PR[GP1:91,2] = PR[GP1:90,2] + 34.694;
   1:L PR[91] R[100]mm/sec CNT100;
   1:  PR[GP1:91,1] = PR[GP1:90,1] + 36.404;
   1:  PR[GP1:91,2] = PR[GP1:90,2] + 34.570;
   1:L PR[91] R[100]mm/sec CNT100;
   1:  PR[GP1:91,1] = PR[GP1:90,1] + 27.653;
   1:  PR[GP1:91,2] = PR[GP1:90,2] + 33.281;
   1:L PR[91] R[100]mm/sec CNT100;
   1:  PR[GP1:91,1] = PR[GP1:90,1] + 23.916;
   1:  PR[GP1:91,2] = PR[GP1:90,2] + 31.863;
   1:L PR[91] R[100]mm/sec CNT100;
   1:  PR[GP1:91,1] = PR[GP1:90,1] + 18.200;
   1:  PR[GP1:91,2] = PR[GP1:90,2] + 29.076;
   1:L PR[91] R[100]mm/sec CNT100;
   1:  PR[GP1:91,1] = PR[GP1:90,1] + 13.332;
   1:  PR[GP1:91,2] = PR[GP1:90,2] + 25.313;
   1:L PR[91] R[100]mm/sec CNT100;
   1:  PR[GP1:91,1] = PR[GP1:90,1] + 10.463;
   1:  PR[GP1:91,2] = PR[GP1:90,2] + 22.534;
   1:L PR[91] R[100]mm/sec CNT100;
   1:  PR[GP1:91,1] = PR[GP1:90,1] + 5.776;
   1:  PR[GP1:91,2] = PR[GP1:90,2] + 15.745;
   1:L PR[91] R[100]mm/sec CNT100;
   1:  PR[GP1:91,1] = PR[GP1:90,1] + 4.892;
   1:  PR[GP1:91,2] = PR[GP1:90,2] + 14.063;
   1:L PR[91] R[100]mm/sec CNT100;
   1:  PR[GP1:91,1] = PR[GP1:90,1] + 3.426;
   1:  PR[GP1:91,2] = PR[GP1:90,2] + 12.489;
   1:L PR[91] R[100]mm/sec CNT100;
   1:  PR[GP1:91,1] = PR[GP1:90,1] + 2.424;
   1:  PR[GP1:91,2] = PR[GP1:90,2] + 11.386;
   1:L PR[91] R[100]mm/sec CNT100;
   1:  PR[GP1:91,1] = PR[GP1:90,1] + 1.857;
   1:  PR[GP1:91,2] = PR[GP1:90,2] + 11.055;
   1:L PR[91] R[100]mm/sec CNT100;
   1:  PR[GP1:91,1] = PR[GP1:90,1] + -1.719;
   1:  PR[GP1:91,2] = PR[GP1:90,2] + 11.090;
   1:L PR[91] R[100]mm/sec CNT100;
   1:  ! -- Layer/Ebene 47 -- !;
   1:  PR[91] = PR[90];
   1:  PR[GP1:91,1] = PR[GP1:90,1] + -2.405;
   1:  PR[GP1:91,2] = PR[GP1:90,2] + 11.973;
   1:  PR[GP1:91,3] = PR[GP1:90,3] + 28.975;
   1:L PR[91] R[100]mm/sec CNT100;
   1:  PR[GP1:91,1] = PR[GP1:90,1] + -4.722;
   1:  PR[GP1:91,2] = PR[GP1:90,2] + 14.473;
   1:L PR[91] R[100]mm/sec CNT100;
   1:  PR[GP1:91,1] = PR[GP1:90,1] + -4.741;
   1:  PR[GP1:91,2] = PR[GP1:90,2] + 14.644;
   1:L PR[91] R[100]mm/sec CNT100;
   1:  PR[GP1:91,1] = PR[GP1:90,1] + -5.059;
   1:  PR[GP1:91,2] = PR[GP1:90,2] + 15.251;
   1:L PR[91] R[100]mm/sec CNT100;
   1:  PR[GP1:91,1] = PR[GP1:90,1] + -10.298;
   1:  PR[GP1:91,2] = PR[GP1:90,2] + 22.837;
   1:L PR[91] R[100]mm/sec CNT100;
   1:  PR[GP1:91,1] = PR[GP1:90,1] + -12.472;
   1:  PR[GP1:91,2] = PR[GP1:90,2] + 24.937;
   1:L PR[91] R[100]mm/sec CNT100;
   1:  PR[GP1:91,1] = PR[GP1:90,1] + -18.067;
   1:  PR[GP1:91,2] = PR[GP1:90,2] + 29.256;
   1:L PR[91] R[100]mm/sec CNT100;
   1:  PR[GP1:91,1] = PR[GP1:90,1] + -22.951;
   1:  PR[GP1:91,2] = PR[GP1:90,2] + 31.639;
   1:L PR[91] R[100]mm/sec CNT100;
   1:  PR[GP1:91,1] = PR[GP1:90,1] + -27.514;
   1:  PR[GP1:91,2] = PR[GP1:90,2] + 33.373;
   1:L PR[91] R[100]mm/sec CNT100;
   1:  PR[GP1:91,1] = PR[GP1:90,1] + -35.402;
   1:  PR[GP1:91,2] = PR[GP1:90,2] + 34.530;
   1:L PR[91] R[100]mm/sec CNT100;
   1:  PR[GP1:91,1] = PR[GP1:90,1] + -37.981;
   1:  PR[GP1:91,2] = PR[GP1:90,2] + 34.714;
   1:L PR[91] R[100]mm/sec CNT100;
   1:  PR[GP1:91,1] = PR[GP1:90,1] + -48.105;
   1:  PR[GP1:91,2] = PR[GP1:90,2] + 33.082;
   1:L PR[91] R[100]mm/sec CNT100;
   1:  PR[GP1:91,1] = PR[GP1:90,1] + -48.604;
   1:  PR[GP1:91,2] = PR[GP1:90,2] + 32.971;
   1:L PR[91] R[100]mm/sec CNT100;
   1:  PR[GP1:91,1] = PR[GP1:90,1] + -58.308;
   1:  PR[GP1:91,2] = PR[GP1:90,2] + 28.113;
   1:L PR[91] R[100]mm/sec CNT100;
   1:  PR[GP1:91,1] = PR[GP1:90,1] + -58.958;
   1:  PR[GP1:91,2] = PR[GP1:90,2] + 27.520;
   1:L PR[91] R[100]mm/sec CNT100;
   1:  PR[GP1:91,1] = PR[GP1:90,1] + -66.094;
   1:  PR[GP1:91,2] = PR[GP1:90,2] + 20.497;
   1:L PR[91] R[100]mm/sec CNT100;
   1:  PR[GP1:91,1] = PR[GP1:90,1] + -67.024;
   1:  PR[GP1:91,2] = PR[GP1:90,2] + 18.794;
   1:L PR[91] R[100]mm/sec CNT100;
   1:  PR[GP1:91,1] = PR[GP1:90,1] + -71.165;
   1:  PR[GP1:91,2] = PR[GP1:90,2] + 10.780;
   1:L PR[91] R[100]mm/sec CNT100;
   1:  PR[GP1:91,1] = PR[GP1:90,1] + -71.598;
   1:  PR[GP1:91,2] = PR[GP1:90,2] + 8.220;
   1:L PR[91] R[100]mm/sec CNT100;
   1:  PR[GP1:91,1] = PR[GP1:90,1] + -72.927;
   1:  PR[GP1:91,2] = PR[GP1:90,2] + -0.069;
   1:L PR[91] R[100]mm/sec CNT100;
   1:  PR[GP1:91,1] = PR[GP1:90,1] + -72.473;
   1:  PR[GP1:91,2] = PR[GP1:90,2] + -2.747;
   1:L PR[91] R[100]mm/sec CNT100;
   1:  PR[GP1:91,1] = PR[GP1:90,1] + -71.164;
   1:  PR[GP1:91,2] = PR[GP1:90,2] + -10.927;
   1:L PR[91] R[100]mm/sec CNT100;
   1:  PR[GP1:91,1] = PR[GP1:90,1] + -67.024;
   1:  PR[GP1:91,2] = PR[GP1:90,2] + -18.938;
   1:L PR[91] R[100]mm/sec CNT100;
   1:  PR[GP1:91,1] = PR[GP1:90,1] + -66.094;
   1:  PR[GP1:91,2] = PR[GP1:90,2] + -20.641;
   1:L PR[91] R[100]mm/sec CNT100;
   1:  PR[GP1:91,1] = PR[GP1:90,1] + -58.958;
   1:  PR[GP1:91,2] = PR[GP1:90,2] + -27.664;
   1:L PR[91] R[100]mm/sec CNT100;
   1:  PR[GP1:91,1] = PR[GP1:90,1] + -58.308;
   1:  PR[GP1:91,2] = PR[GP1:90,2] + -28.257;
   1:L PR[91] R[100]mm/sec CNT100;
   1:  PR[GP1:91,1] = PR[GP1:90,1] + -48.605;
   1:  PR[GP1:91,2] = PR[GP1:90,2] + -33.115;
   1:L PR[91] R[100]mm/sec CNT100;
   1:  PR[GP1:91,1] = PR[GP1:90,1] + -48.106;
   1:  PR[GP1:91,2] = PR[GP1:90,2] + -33.226;
   1:L PR[91] R[100]mm/sec CNT100;
   1:  PR[GP1:91,1] = PR[GP1:90,1] + -37.981;
   1:  PR[GP1:91,2] = PR[GP1:90,2] + -34.858;
   1:L PR[91] R[100]mm/sec CNT100;
   1:  PR[GP1:91,1] = PR[GP1:90,1] + -35.402;
   1:  PR[GP1:91,2] = PR[GP1:90,2] + -34.674;
   1:L PR[91] R[100]mm/sec CNT100;
   1:  PR[GP1:91,1] = PR[GP1:90,1] + -27.514;
   1:  PR[GP1:91,2] = PR[GP1:90,2] + -33.517;
   1:L PR[91] R[100]mm/sec CNT100;
   1:  PR[GP1:91,1] = PR[GP1:90,1] + -22.951;
   1:  PR[GP1:91,2] = PR[GP1:90,2] + -31.783;
   1:L PR[91] R[100]mm/sec CNT100;
   1:  PR[GP1:91,1] = PR[GP1:90,1] + -18.067;
   1:  PR[GP1:91,2] = PR[GP1:90,2] + -29.400;
   1:L PR[91] R[100]mm/sec CNT100;
   1:  PR[GP1:91,1] = PR[GP1:90,1] + -12.472;
   1:  PR[GP1:91,2] = PR[GP1:90,2] + -25.081;
   1:L PR[91] R[100]mm/sec CNT100;
   1:  PR[GP1:91,1] = PR[GP1:90,1] + -10.298;
   1:  PR[GP1:91,2] = PR[GP1:90,2] + -22.981;
   1:L PR[91] R[100]mm/sec CNT100;
   1:  PR[GP1:91,1] = PR[GP1:90,1] + -5.039;
   1:  PR[GP1:91,2] = PR[GP1:90,2] + -15.356;
   1:L PR[91] R[100]mm/sec CNT100;
   1:  PR[GP1:91,1] = PR[GP1:90,1] + -4.654;
   1:  PR[GP1:91,2] = PR[GP1:90,2] + -14.618;
   1:L PR[91] R[100]mm/sec CNT100;
   1:  PR[GP1:91,1] = PR[GP1:90,1] + -2.410;
   1:  PR[GP1:91,2] = PR[GP1:90,2] + -12.120;
   1:L PR[91] R[100]mm/sec CNT100;
   1:  PR[GP1:91,1] = PR[GP1:90,1] + -1.616;
   1:  PR[GP1:91,2] = PR[GP1:90,2] + -11.656;
   1:L PR[91] R[100]mm/sec CNT100;
   1:  PR[GP1:91,1] = PR[GP1:90,1] + 1.878;
   1:  PR[GP1:91,2] = PR[GP1:90,2] + -11.621;
   1:L PR[91] R[100]mm/sec CNT100;
   1:  PR[GP1:91,1] = PR[GP1:90,1] + 3.742;
   1:  PR[GP1:91,2] = PR[GP1:90,2] + -13.855;
   1:L PR[91] R[100]mm/sec CNT100;
   1:  PR[GP1:91,1] = PR[GP1:90,1] + 4.822;
   1:  PR[GP1:91,2] = PR[GP1:90,2] + -14.536;
   1:L PR[91] R[100]mm/sec CNT100;
   1:  PR[GP1:91,1] = PR[GP1:90,1] + 5.244;
   1:  PR[GP1:91,2] = PR[GP1:90,2] + -15.339;
   1:L PR[91] R[100]mm/sec CNT100;
   1:  PR[GP1:91,1] = PR[GP1:90,1] + 10.509;
   1:  PR[GP1:91,2] = PR[GP1:90,2] + -22.972;
   1:L PR[91] R[100]mm/sec CNT100;
   1:  PR[GP1:91,1] = PR[GP1:90,1] + 12.681;
   1:  PR[GP1:91,2] = PR[GP1:90,2] + -25.076;
   1:L PR[91] R[100]mm/sec CNT100;
   1:  PR[GP1:91,1] = PR[GP1:90,1] + 18.275;
   1:  PR[GP1:91,2] = PR[GP1:90,2] + -29.400;
   1:L PR[91] R[100]mm/sec CNT100;
   1:  PR[GP1:91,1] = PR[GP1:90,1] + 23.157;
   1:  PR[GP1:91,2] = PR[GP1:90,2] + -31.781;
   1:L PR[91] R[100]mm/sec CNT100;
   1:  PR[GP1:91,1] = PR[GP1:90,1] + 27.719;
   1:  PR[GP1:91,2] = PR[GP1:90,2] + -33.513;
   1:L PR[91] R[100]mm/sec CNT100;
   1:  PR[GP1:91,1] = PR[GP1:90,1] + 35.605;
   1:  PR[GP1:91,2] = PR[GP1:90,2] + -34.674;
   1:L PR[91] R[100]mm/sec CNT100;
   1:  PR[GP1:91,1] = PR[GP1:90,1] + 38.185;
   1:  PR[GP1:91,2] = PR[GP1:90,2] + -34.858;
   1:L PR[91] R[100]mm/sec CNT100;
   1:  PR[GP1:91,1] = PR[GP1:90,1] + 48.309;
   1:  PR[GP1:91,2] = PR[GP1:90,2] + -33.227;
   1:L PR[91] R[100]mm/sec CNT100;
   1:  PR[GP1:91,1] = PR[GP1:90,1] + 48.809;
   1:  PR[GP1:91,2] = PR[GP1:90,2] + -33.115;
   1:L PR[91] R[100]mm/sec CNT100;
   1:  PR[GP1:91,1] = PR[GP1:90,1] + 58.516;
   1:  PR[GP1:91,2] = PR[GP1:90,2] + -28.264;
   1:L PR[91] R[100]mm/sec CNT100;
   1:  PR[GP1:91,1] = PR[GP1:90,1] + 59.166;
   1:  PR[GP1:91,2] = PR[GP1:90,2] + -27.671;
   1:L PR[91] R[100]mm/sec CNT100;
   1:  PR[GP1:91,1] = PR[GP1:90,1] + 66.304;
   1:  PR[GP1:91,2] = PR[GP1:90,2] + -20.636;
   1:L PR[91] R[100]mm/sec CNT100;
   1:  PR[GP1:91,1] = PR[GP1:90,1] + 67.235;
   1:  PR[GP1:91,2] = PR[GP1:90,2] + -18.934;
   1:L PR[91] R[100]mm/sec CNT100;
   1:  PR[GP1:91,1] = PR[GP1:90,1] + 71.378;
   1:  PR[GP1:91,2] = PR[GP1:90,2] + -10.939;
   1:L PR[91] R[100]mm/sec CNT100;
   1:  PR[GP1:91,1] = PR[GP1:90,1] + 71.811;
   1:  PR[GP1:91,2] = PR[GP1:90,2] + -8.378;
   1:L PR[91] R[100]mm/sec CNT100;
   1:  PR[GP1:91,1] = PR[GP1:90,1] + 73.140;
   1:  PR[GP1:91,2] = PR[GP1:90,2] + -0.075;
   1:L PR[91] R[100]mm/sec CNT100;
   1:  PR[GP1:91,1] = PR[GP1:90,1] + 72.686;
   1:  PR[GP1:91,2] = PR[GP1:90,2] + 2.605;
   1:L PR[91] R[100]mm/sec CNT100;
   1:  PR[GP1:91,1] = PR[GP1:90,1] + 71.376;
   1:  PR[GP1:91,2] = PR[GP1:90,2] + 10.798;
   1:L PR[91] R[100]mm/sec CNT100;
   1:  PR[GP1:91,1] = PR[GP1:90,1] + 67.235;
   1:  PR[GP1:91,2] = PR[GP1:90,2] + 18.790;
   1:L PR[91] R[100]mm/sec CNT100;
   1:  PR[GP1:91,1] = PR[GP1:90,1] + 66.304;
   1:  PR[GP1:91,2] = PR[GP1:90,2] + 20.492;
   1:L PR[91] R[100]mm/sec CNT100;
   1:  PR[GP1:91,1] = PR[GP1:90,1] + 59.166;
   1:  PR[GP1:91,2] = PR[GP1:90,2] + 27.527;
   1:L PR[91] R[100]mm/sec CNT100;
   1:  PR[GP1:91,1] = PR[GP1:90,1] + 58.516;
   1:  PR[GP1:91,2] = PR[GP1:90,2] + 28.120;
   1:L PR[91] R[100]mm/sec CNT100;
   1:  PR[GP1:91,1] = PR[GP1:90,1] + 48.809;
   1:  PR[GP1:91,2] = PR[GP1:90,2] + 32.971;
   1:L PR[91] R[100]mm/sec CNT100;
   1:  PR[GP1:91,1] = PR[GP1:90,1] + 48.309;
   1:  PR[GP1:91,2] = PR[GP1:90,2] + 33.083;
   1:L PR[91] R[100]mm/sec CNT100;
   1:  PR[GP1:91,1] = PR[GP1:90,1] + 38.185;
   1:  PR[GP1:91,2] = PR[GP1:90,2] + 34.714;
   1:L PR[91] R[100]mm/sec CNT100;
   1:  PR[GP1:91,1] = PR[GP1:90,1] + 35.605;
   1:  PR[GP1:91,2] = PR[GP1:90,2] + 34.530;
   1:L PR[91] R[100]mm/sec CNT100;
   1:  PR[GP1:91,1] = PR[GP1:90,1] + 27.719;
   1:  PR[GP1:91,2] = PR[GP1:90,2] + 33.369;
   1:L PR[91] R[100]mm/sec CNT100;
   1:  PR[GP1:91,1] = PR[GP1:90,1] + 23.157;
   1:  PR[GP1:91,2] = PR[GP1:90,2] + 31.637;
   1:L PR[91] R[100]mm/sec CNT100;
   1:  PR[GP1:91,1] = PR[GP1:90,1] + 18.275;
   1:  PR[GP1:91,2] = PR[GP1:90,2] + 29.256;
   1:L PR[91] R[100]mm/sec CNT100;
   1:  PR[GP1:91,1] = PR[GP1:90,1] + 12.681;
   1:  PR[GP1:91,2] = PR[GP1:90,2] + 24.932;
   1:L PR[91] R[100]mm/sec CNT100;
   1:  PR[GP1:91,1] = PR[GP1:90,1] + 10.508;
   1:  PR[GP1:91,2] = PR[GP1:90,2] + 22.828;
   1:L PR[91] R[100]mm/sec CNT100;
   1:  PR[GP1:91,1] = PR[GP1:90,1] + 5.265;
   1:  PR[GP1:91,2] = PR[GP1:90,2] + 15.235;
   1:L PR[91] R[100]mm/sec CNT100;
   1:  PR[GP1:91,1] = PR[GP1:90,1] + 4.861;
   1:  PR[GP1:91,2] = PR[GP1:90,2] + 14.466;
   1:L PR[91] R[100]mm/sec CNT100;
   1:  PR[GP1:91,1] = PR[GP1:90,1] + 2.552;
   1:  PR[GP1:91,2] = PR[GP1:90,2] + 11.942;
   1:L PR[91] R[100]mm/sec CNT100;
   1:  PR[GP1:91,1] = PR[GP1:90,1] + 1.759;
   1:  PR[GP1:91,2] = PR[GP1:90,2] + 11.479;
   1:L PR[91] R[100]mm/sec CNT100;
   1:  PR[GP1:91,1] = PR[GP1:90,1] + -1.616;
   1:  PR[GP1:91,2] = PR[GP1:90,2] + 11.511;
   1:L PR[91] R[100]mm/sec CNT100;
   1:  ! -- Layer/Ebene 48 -- !;
   1:  PR[91] = PR[90];
   1:  PR[GP1:91,1] = PR[GP1:90,1] + -2.528;
   1:  PR[GP1:91,2] = PR[GP1:90,2] + 12.528;
   1:  PR[GP1:91,3] = PR[GP1:90,3] + 29.585;
   1:L PR[91] R[100]mm/sec CNT100;
   1:  PR[GP1:91,1] = PR[GP1:90,1] + -4.688;
   1:  PR[GP1:91,2] = PR[GP1:90,2] + 14.857;
   1:L PR[91] R[100]mm/sec CNT100;
   1:  PR[GP1:91,1] = PR[GP1:90,1] + -4.703;
   1:  PR[GP1:91,2] = PR[GP1:90,2] + 14.993;
   1:L PR[91] R[100]mm/sec CNT100;
   1:  PR[GP1:91,1] = PR[GP1:90,1] + -5.082;
   1:  PR[GP1:91,2] = PR[GP1:90,2] + 15.511;
   1:L PR[91] R[100]mm/sec CNT100;
   1:  PR[GP1:91,1] = PR[GP1:90,1] + -10.342;
   1:  PR[GP1:91,2] = PR[GP1:90,2] + 23.129;
   1:L PR[91] R[100]mm/sec CNT100;
   1:  PR[GP1:91,1] = PR[GP1:90,1] + -11.819;
   1:  PR[GP1:91,2] = PR[GP1:90,2] + 24.556;
   1:L PR[91] R[100]mm/sec CNT100;
   1:  PR[GP1:91,1] = PR[GP1:90,1] + -18.140;
   1:  PR[GP1:91,2] = PR[GP1:90,2] + 29.436;
   1:L PR[91] R[100]mm/sec CNT100;
   1:  PR[GP1:91,1] = PR[GP1:90,1] + -22.191;
   1:  PR[GP1:91,2] = PR[GP1:90,2] + 31.412;
   1:L PR[91] R[100]mm/sec CNT100;
   1:  PR[GP1:91,1] = PR[GP1:90,1] + -27.579;
   1:  PR[GP1:91,2] = PR[GP1:90,2] + 33.460;
   1:L PR[91] R[100]mm/sec CNT100;
   1:  PR[GP1:91,1] = PR[GP1:90,1] + -34.602;
   1:  PR[GP1:91,2] = PR[GP1:90,2] + 34.491;
   1:L PR[91] R[100]mm/sec CNT100;
   1:  PR[GP1:91,1] = PR[GP1:90,1] + -38.015;
   1:  PR[GP1:91,2] = PR[GP1:90,2] + 34.733;
   1:L PR[91] R[100]mm/sec CNT100;
   1:  PR[GP1:91,1] = PR[GP1:90,1] + -47.337;
   1:  PR[GP1:91,2] = PR[GP1:90,2] + 33.231;
   1:L PR[91] R[100]mm/sec CNT100;
   1:  PR[GP1:91,1] = PR[GP1:90,1] + -48.596;
   1:  PR[GP1:91,2] = PR[GP1:90,2] + 32.949;
   1:L PR[91] R[100]mm/sec CNT100;
   1:  PR[GP1:91,1] = PR[GP1:90,1] + -58.316;
   1:  PR[GP1:91,2] = PR[GP1:90,2] + 28.068;
   1:L PR[91] R[100]mm/sec CNT100;
   1:  PR[GP1:91,1] = PR[GP1:90,1] + -58.459;
   1:  PR[GP1:91,2] = PR[GP1:90,2] + 27.937;
   1:L PR[91] R[100]mm/sec CNT100;
   1:  PR[GP1:91,1] = PR[GP1:90,1] + -66.063;
   1:  PR[GP1:91,2] = PR[GP1:90,2] + 20.454;
   1:L PR[91] R[100]mm/sec CNT100;
   1:  PR[GP1:91,1] = PR[GP1:90,1] + -66.684;
   1:  PR[GP1:91,2] = PR[GP1:90,2] + 19.317;
   1:L PR[91] R[100]mm/sec CNT100;
   1:  PR[GP1:91,1] = PR[GP1:90,1] + -71.108;
   1:  PR[GP1:91,2] = PR[GP1:90,2] + 10.755;
   1:L PR[91] R[100]mm/sec CNT100;
   1:  PR[GP1:91,1] = PR[GP1:90,1] + -71.436;
   1:  PR[GP1:91,2] = PR[GP1:90,2] + 8.817;
   1:L PR[91] R[100]mm/sec CNT100;
   1:  PR[GP1:91,1] = PR[GP1:90,1] + -72.861;
   1:  PR[GP1:91,2] = PR[GP1:90,2] + -0.069;
   1:L PR[91] R[100]mm/sec CNT100;
   1:  PR[GP1:91,1] = PR[GP1:90,1] + -72.506;
   1:  PR[GP1:91,2] = PR[GP1:90,2] + -2.162;
   1:L PR[91] R[100]mm/sec CNT100;
   1:  PR[GP1:91,1] = PR[GP1:90,1] + -71.107;
   1:  PR[GP1:91,2] = PR[GP1:90,2] + -10.901;
   1:L PR[91] R[100]mm/sec CNT100;
   1:  PR[GP1:91,1] = PR[GP1:90,1] + -66.684;
   1:  PR[GP1:91,2] = PR[GP1:90,2] + -19.461;
   1:L PR[91] R[100]mm/sec CNT100;
   1:  PR[GP1:91,1] = PR[GP1:90,1] + -66.063;
   1:  PR[GP1:91,2] = PR[GP1:90,2] + -20.598;
   1:L PR[91] R[100]mm/sec CNT100;
   1:  PR[GP1:91,1] = PR[GP1:90,1] + -58.459;
   1:  PR[GP1:91,2] = PR[GP1:90,2] + -28.081;
   1:L PR[91] R[100]mm/sec CNT100;
   1:  PR[GP1:91,1] = PR[GP1:90,1] + -58.316;
   1:  PR[GP1:91,2] = PR[GP1:90,2] + -28.212;
   1:L PR[91] R[100]mm/sec CNT100;
   1:  PR[GP1:91,1] = PR[GP1:90,1] + -48.596;
   1:  PR[GP1:91,2] = PR[GP1:90,2] + -33.093;
   1:L PR[91] R[100]mm/sec CNT100;
   1:  PR[GP1:91,1] = PR[GP1:90,1] + -47.337;
   1:  PR[GP1:91,2] = PR[GP1:90,2] + -33.375;
   1:L PR[91] R[100]mm/sec CNT100;
   1:  PR[GP1:91,1] = PR[GP1:90,1] + -38.015;
   1:  PR[GP1:91,2] = PR[GP1:90,2] + -34.877;
   1:L PR[91] R[100]mm/sec CNT100;
   1:  PR[GP1:91,1] = PR[GP1:90,1] + -34.602;
   1:  PR[GP1:91,2] = PR[GP1:90,2] + -34.635;
   1:L PR[91] R[100]mm/sec CNT100;
   1:  PR[GP1:91,1] = PR[GP1:90,1] + -27.579;
   1:  PR[GP1:91,2] = PR[GP1:90,2] + -33.605;
   1:L PR[91] R[100]mm/sec CNT100;
   1:  PR[GP1:91,1] = PR[GP1:90,1] + -22.191;
   1:  PR[GP1:91,2] = PR[GP1:90,2] + -31.556;
   1:L PR[91] R[100]mm/sec CNT100;
   1:  PR[GP1:91,1] = PR[GP1:90,1] + -18.140;
   1:  PR[GP1:91,2] = PR[GP1:90,2] + -29.580;
   1:L PR[91] R[100]mm/sec CNT100;
   1:  PR[GP1:91,1] = PR[GP1:90,1] + -11.819;
   1:  PR[GP1:91,2] = PR[GP1:90,2] + -24.700;
   1:L PR[91] R[100]mm/sec CNT100;
   1:  PR[GP1:91,1] = PR[GP1:90,1] + -10.342;
   1:  PR[GP1:91,2] = PR[GP1:90,2] + -23.273;
   1:L PR[91] R[100]mm/sec CNT100;
   1:  PR[GP1:91,1] = PR[GP1:90,1] + -5.186;
   1:  PR[GP1:91,2] = PR[GP1:90,2] + -15.797;
   1:L PR[91] R[100]mm/sec CNT100;
   1:  PR[GP1:91,1] = PR[GP1:90,1] + -4.591;
   1:  PR[GP1:91,2] = PR[GP1:90,2] + -14.984;
   1:L PR[91] R[100]mm/sec CNT100;
   1:  PR[GP1:91,1] = PR[GP1:90,1] + -2.533;
   1:  PR[GP1:91,2] = PR[GP1:90,2] + -12.675;
   1:L PR[91] R[100]mm/sec CNT100;
   1:  PR[GP1:91,1] = PR[GP1:90,1] + -1.512;
   1:  PR[GP1:91,2] = PR[GP1:90,2] + -12.077;
   1:L PR[91] R[100]mm/sec CNT100;
   1:  PR[GP1:91,1] = PR[GP1:90,1] + 1.779;
   1:  PR[GP1:91,2] = PR[GP1:90,2] + -12.045;
   1:L PR[91] R[100]mm/sec CNT100;
   1:  PR[GP1:91,1] = PR[GP1:90,1] + 3.528;
   1:  PR[GP1:91,2] = PR[GP1:90,2] + -14.140;
   1:L PR[91] R[100]mm/sec CNT100;
   1:  PR[GP1:91,1] = PR[GP1:90,1] + 4.750;
   1:  PR[GP1:91,2] = PR[GP1:90,2] + -14.905;
   1:L PR[91] R[100]mm/sec CNT100;
   1:  PR[GP1:91,1] = PR[GP1:90,1] + 5.408;
   1:  PR[GP1:91,2] = PR[GP1:90,2] + -15.806;
   1:L PR[91] R[100]mm/sec CNT100;
   1:  PR[GP1:91,1] = PR[GP1:90,1] + 10.553;
   1:  PR[GP1:91,2] = PR[GP1:90,2] + -23.266;
   1:L PR[91] R[100]mm/sec CNT100;
   1:  PR[GP1:91,1] = PR[GP1:90,1] + 12.030;
   1:  PR[GP1:91,2] = PR[GP1:90,2] + -24.696;
   1:L PR[91] R[100]mm/sec CNT100;
   1:  PR[GP1:91,1] = PR[GP1:90,1] + 18.349;
   1:  PR[GP1:91,2] = PR[GP1:90,2] + -29.581;
   1:L PR[91] R[100]mm/sec CNT100;
   1:  PR[GP1:91,1] = PR[GP1:90,1] + 22.398;
   1:  PR[GP1:91,2] = PR[GP1:90,2] + -31.555;
   1:L PR[91] R[100]mm/sec CNT100;
   1:  PR[GP1:91,1] = PR[GP1:90,1] + 27.785;
   1:  PR[GP1:91,2] = PR[GP1:90,2] + -33.600;
   1:L PR[91] R[100]mm/sec CNT100;
   1:  PR[GP1:91,1] = PR[GP1:90,1] + 34.807;
   1:  PR[GP1:91,2] = PR[GP1:90,2] + -34.634;
   1:L PR[91] R[100]mm/sec CNT100;
   1:  PR[GP1:91,1] = PR[GP1:90,1] + 38.220;
   1:  PR[GP1:91,2] = PR[GP1:90,2] + -34.878;
   1:L PR[91] R[100]mm/sec CNT100;
   1:  PR[GP1:91,1] = PR[GP1:90,1] + 47.541;
   1:  PR[GP1:91,2] = PR[GP1:90,2] + -33.376;
   1:L PR[91] R[100]mm/sec CNT100;
   1:  PR[GP1:91,1] = PR[GP1:90,1] + 48.802;
   1:  PR[GP1:91,2] = PR[GP1:90,2] + -33.094;
   1:L PR[91] R[100]mm/sec CNT100;
   1:  PR[GP1:91,1] = PR[GP1:90,1] + 58.524;
   1:  PR[GP1:91,2] = PR[GP1:90,2] + -28.219;
   1:L PR[91] R[100]mm/sec CNT100;
   1:  PR[GP1:91,1] = PR[GP1:90,1] + 58.666;
   1:  PR[GP1:91,2] = PR[GP1:90,2] + -28.089;
   1:L PR[91] R[100]mm/sec CNT100;
   1:  PR[GP1:91,1] = PR[GP1:90,1] + 66.273;
   1:  PR[GP1:91,2] = PR[GP1:90,2] + -20.593;
   1:L PR[91] R[100]mm/sec CNT100;
   1:  PR[GP1:91,1] = PR[GP1:90,1] + 66.894;
   1:  PR[GP1:91,2] = PR[GP1:90,2] + -19.456;
   1:L PR[91] R[100]mm/sec CNT100;
   1:  PR[GP1:91,1] = PR[GP1:90,1] + 71.321;
   1:  PR[GP1:91,2] = PR[GP1:90,2] + -10.915;
   1:L PR[91] R[100]mm/sec CNT100;
   1:  PR[GP1:91,1] = PR[GP1:90,1] + 71.649;
   1:  PR[GP1:91,2] = PR[GP1:90,2] + -8.976;
   1:L PR[91] R[100]mm/sec CNT100;
   1:  PR[GP1:91,1] = PR[GP1:90,1] + 73.074;
   1:  PR[GP1:91,2] = PR[GP1:90,2] + -0.075;
   1:L PR[91] R[100]mm/sec CNT100;
   1:  PR[GP1:91,1] = PR[GP1:90,1] + 72.719;
   1:  PR[GP1:91,2] = PR[GP1:90,2] + 2.019;
   1:L PR[91] R[100]mm/sec CNT100;
   1:  PR[GP1:91,1] = PR[GP1:90,1] + 71.320;
   1:  PR[GP1:91,2] = PR[GP1:90,2] + 10.773;
   1:L PR[91] R[100]mm/sec CNT100;
   1:  PR[GP1:91,1] = PR[GP1:90,1] + 66.894;
   1:  PR[GP1:91,2] = PR[GP1:90,2] + 19.312;
   1:L PR[91] R[100]mm/sec CNT100;
   1:  PR[GP1:91,1] = PR[GP1:90,1] + 66.273;
   1:  PR[GP1:91,2] = PR[GP1:90,2] + 20.449;
   1:L PR[91] R[100]mm/sec CNT100;
   1:  PR[GP1:91,1] = PR[GP1:90,1] + 58.666;
   1:  PR[GP1:91,2] = PR[GP1:90,2] + 27.945;
   1:L PR[91] R[100]mm/sec CNT100;
   1:  PR[GP1:91,1] = PR[GP1:90,1] + 58.524;
   1:  PR[GP1:91,2] = PR[GP1:90,2] + 28.075;
   1:L PR[91] R[100]mm/sec CNT100;
   1:  PR[GP1:91,1] = PR[GP1:90,1] + 48.802;
   1:  PR[GP1:91,2] = PR[GP1:90,2] + 32.950;
   1:L PR[91] R[100]mm/sec CNT100;
   1:  PR[GP1:91,1] = PR[GP1:90,1] + 47.541;
   1:  PR[GP1:91,2] = PR[GP1:90,2] + 33.232;
   1:L PR[91] R[100]mm/sec CNT100;
   1:  PR[GP1:91,1] = PR[GP1:90,1] + 38.220;
   1:  PR[GP1:91,2] = PR[GP1:90,2] + 34.734;
   1:L PR[91] R[100]mm/sec CNT100;
   1:  PR[GP1:91,1] = PR[GP1:90,1] + 34.807;
   1:  PR[GP1:91,2] = PR[GP1:90,2] + 34.490;
   1:L PR[91] R[100]mm/sec CNT100;
   1:  PR[GP1:91,1] = PR[GP1:90,1] + 27.785;
   1:  PR[GP1:91,2] = PR[GP1:90,2] + 33.456;
   1:L PR[91] R[100]mm/sec CNT100;
   1:  PR[GP1:91,1] = PR[GP1:90,1] + 22.398;
   1:  PR[GP1:91,2] = PR[GP1:90,2] + 31.411;
   1:L PR[91] R[100]mm/sec CNT100;
   1:  PR[GP1:91,1] = PR[GP1:90,1] + 18.349;
   1:  PR[GP1:91,2] = PR[GP1:90,2] + 29.437;
   1:L PR[91] R[100]mm/sec CNT100;
   1:  PR[GP1:91,1] = PR[GP1:90,1] + 12.030;
   1:  PR[GP1:91,2] = PR[GP1:90,2] + 24.552;
   1:L PR[91] R[100]mm/sec CNT100;
   1:  PR[GP1:91,1] = PR[GP1:90,1] + 10.553;
   1:  PR[GP1:91,2] = PR[GP1:90,2] + 23.122;
   1:L PR[91] R[100]mm/sec CNT100;
   1:  PR[GP1:91,1] = PR[GP1:90,1] + 5.304;
   1:  PR[GP1:91,2] = PR[GP1:90,2] + 15.520;
   1:L PR[91] R[100]mm/sec CNT100;
   1:  PR[GP1:91,1] = PR[GP1:90,1] + 4.799;
   1:  PR[GP1:91,2] = PR[GP1:90,2] + 14.829;
   1:L PR[91] R[100]mm/sec CNT100;
   1:  PR[GP1:91,1] = PR[GP1:90,1] + 2.682;
   1:  PR[GP1:91,2] = PR[GP1:90,2] + 12.498;
   1:L PR[91] R[100]mm/sec CNT100;
   1:  PR[GP1:91,1] = PR[GP1:90,1] + 1.660;
   1:  PR[GP1:91,2] = PR[GP1:90,2] + 11.902;
   1:L PR[91] R[100]mm/sec CNT100;
   1:  PR[GP1:91,1] = PR[GP1:90,1] + -1.512;
   1:  PR[GP1:91,2] = PR[GP1:90,2] + 11.933;
   1:L PR[91] R[100]mm/sec CNT100;
   1:  ! -- Layer/Ebene 49 -- !;
   1:  PR[91] = PR[90];
   1:  PR[GP1:91,1] = PR[GP1:90,1] + -2.651;
   1:  PR[GP1:91,2] = PR[GP1:90,2] + 13.082;
   1:  PR[GP1:91,3] = PR[GP1:90,3] + 30.195;
   1:L PR[91] R[100]mm/sec CNT100;
   1:  PR[GP1:91,1] = PR[GP1:90,1] + -4.653;
   1:  PR[GP1:91,2] = PR[GP1:90,2] + 15.242;
   1:L PR[91] R[100]mm/sec CNT100;
   1:  PR[GP1:91,1] = PR[GP1:90,1] + -4.667;
   1:  PR[GP1:91,2] = PR[GP1:90,2] + 15.370;
   1:L PR[91] R[100]mm/sec CNT100;
   1:  PR[GP1:91,1] = PR[GP1:90,1] + -7.511;
   1:  PR[GP1:91,2] = PR[GP1:90,2] + 19.259;
   1:L PR[91] R[100]mm/sec CNT100;
   1:  PR[GP1:91,1] = PR[GP1:90,1] + -10.386;
   1:  PR[GP1:91,2] = PR[GP1:90,2] + 23.421;
   1:L PR[91] R[100]mm/sec CNT100;
   1:  PR[GP1:91,1] = PR[GP1:90,1] + -11.167;
   1:  PR[GP1:91,2] = PR[GP1:90,2] + 24.176;
   1:L PR[91] R[100]mm/sec CNT100;
   1:  PR[GP1:91,1] = PR[GP1:90,1] + -18.214;
   1:  PR[GP1:91,2] = PR[GP1:90,2] + 29.616;
   1:L PR[91] R[100]mm/sec CNT100;
   1:  PR[GP1:91,1] = PR[GP1:90,1] + -21.431;
   1:  PR[GP1:91,2] = PR[GP1:90,2] + 31.186;
   1:L PR[91] R[100]mm/sec CNT100;
   1:  PR[GP1:91,1] = PR[GP1:90,1] + -27.645;
   1:  PR[GP1:91,2] = PR[GP1:90,2] + 33.548;
   1:L PR[91] R[100]mm/sec CNT100;
   1:  PR[GP1:91,1] = PR[GP1:90,1] + -33.803;
   1:  PR[GP1:91,2] = PR[GP1:90,2] + 34.451;
   1:L PR[91] R[100]mm/sec CNT100;
   1:  PR[GP1:91,1] = PR[GP1:90,1] + -38.049;
   1:  PR[GP1:91,2] = PR[GP1:90,2] + 34.753;
   1:L PR[91] R[100]mm/sec CNT100;
   1:  PR[GP1:91,1] = PR[GP1:90,1] + -46.568;
   1:  PR[GP1:91,2] = PR[GP1:90,2] + 33.380;
   1:L PR[91] R[100]mm/sec CNT100;
   1:  PR[GP1:91,1] = PR[GP1:90,1] + -48.588;
   1:  PR[GP1:91,2] = PR[GP1:90,2] + 32.928;
   1:L PR[91] R[100]mm/sec CNT100;
   1:  PR[GP1:91,1] = PR[GP1:90,1] + -57.987;
   1:  PR[GP1:91,2] = PR[GP1:90,2] + 28.201;
   1:L PR[91] R[100]mm/sec CNT100;
   1:  PR[GP1:91,1] = PR[GP1:90,1] + -58.270;
   1:  PR[GP1:91,2] = PR[GP1:90,2] + 28.042;
   1:L PR[91] R[100]mm/sec CNT100;
   1:  PR[GP1:91,1] = PR[GP1:90,1] + -66.032;
   1:  PR[GP1:91,2] = PR[GP1:90,2] + 20.411;
   1:L PR[91] R[100]mm/sec CNT100;
   1:  PR[GP1:91,1] = PR[GP1:90,1] + -66.344;
   1:  PR[GP1:91,2] = PR[GP1:90,2] + 19.840;
   1:L PR[91] R[100]mm/sec CNT100;
   1:  PR[GP1:91,1] = PR[GP1:90,1] + -71.051;
   1:  PR[GP1:91,2] = PR[GP1:90,2] + 10.730;
   1:L PR[91] R[100]mm/sec CNT100;
   1:  PR[GP1:91,1] = PR[GP1:90,1] + -71.274;
   1:  PR[GP1:91,2] = PR[GP1:90,2] + 9.413;
   1:L PR[91] R[100]mm/sec CNT100;
   1:  PR[GP1:91,1] = PR[GP1:90,1] + -72.794;
   1:  PR[GP1:91,2] = PR[GP1:90,2] + -0.069;
   1:L PR[91] R[100]mm/sec CNT100;
   1:  PR[GP1:91,1] = PR[GP1:90,1] + -72.538;
   1:  PR[GP1:91,2] = PR[GP1:90,2] + -1.577;
   1:L PR[91] R[100]mm/sec CNT100;
   1:  PR[GP1:91,1] = PR[GP1:90,1] + -71.050;
   1:  PR[GP1:91,2] = PR[GP1:90,2] + -10.876;
   1:L PR[91] R[100]mm/sec CNT100;
   1:  PR[GP1:91,1] = PR[GP1:90,1] + -66.344;
   1:  PR[GP1:91,2] = PR[GP1:90,2] + -19.984;
   1:L PR[91] R[100]mm/sec CNT100;
   1:  PR[GP1:91,1] = PR[GP1:90,1] + -66.032;
   1:  PR[GP1:91,2] = PR[GP1:90,2] + -20.555;
   1:L PR[91] R[100]mm/sec CNT100;
   1:  PR[GP1:91,1] = PR[GP1:90,1] + -58.270;
   1:  PR[GP1:91,2] = PR[GP1:90,2] + -28.186;
   1:L PR[91] R[100]mm/sec CNT100;
   1:  PR[GP1:91,1] = PR[GP1:90,1] + -57.987;
   1:  PR[GP1:91,2] = PR[GP1:90,2] + -28.345;
   1:L PR[91] R[100]mm/sec CNT100;
   1:  PR[GP1:91,1] = PR[GP1:90,1] + -48.588;
   1:  PR[GP1:91,2] = PR[GP1:90,2] + -33.072;
   1:L PR[91] R[100]mm/sec CNT100;
   1:  PR[GP1:91,1] = PR[GP1:90,1] + -46.568;
   1:  PR[GP1:91,2] = PR[GP1:90,2] + -33.524;
   1:L PR[91] R[100]mm/sec CNT100;
   1:  PR[GP1:91,1] = PR[GP1:90,1] + -38.049;
   1:  PR[GP1:91,2] = PR[GP1:90,2] + -34.897;
   1:L PR[91] R[100]mm/sec CNT100;
   1:  PR[GP1:91,1] = PR[GP1:90,1] + -33.803;
   1:  PR[GP1:91,2] = PR[GP1:90,2] + -34.595;
   1:L PR[91] R[100]mm/sec CNT100;
   1:  PR[GP1:91,1] = PR[GP1:90,1] + -27.645;
   1:  PR[GP1:91,2] = PR[GP1:90,2] + -33.692;
   1:L PR[91] R[100]mm/sec CNT100;
   1:  PR[GP1:91,1] = PR[GP1:90,1] + -21.430;
   1:  PR[GP1:91,2] = PR[GP1:90,2] + -31.329;
   1:L PR[91] R[100]mm/sec CNT100;
   1:  PR[GP1:91,1] = PR[GP1:90,1] + -18.213;
   1:  PR[GP1:91,2] = PR[GP1:90,2] + -29.760;
   1:L PR[91] R[100]mm/sec CNT100;
   1:  PR[GP1:91,1] = PR[GP1:90,1] + -11.167;
   1:  PR[GP1:91,2] = PR[GP1:90,2] + -24.320;
   1:L PR[91] R[100]mm/sec CNT100;
   1:  PR[GP1:91,1] = PR[GP1:90,1] + -10.386;
   1:  PR[GP1:91,2] = PR[GP1:90,2] + -23.565;
   1:L PR[91] R[100]mm/sec CNT100;
   1:  PR[GP1:91,1] = PR[GP1:90,1] + -7.569;
   1:  PR[GP1:91,2] = PR[GP1:90,2] + -19.481;
   1:L PR[91] R[100]mm/sec CNT100;
   1:  PR[GP1:91,1] = PR[GP1:90,1] + -4.556;
   1:  PR[GP1:91,2] = PR[GP1:90,2] + -15.361;
   1:L PR[91] R[100]mm/sec CNT100;
   1:  PR[GP1:91,1] = PR[GP1:90,1] + -2.656;
   1:  PR[GP1:91,2] = PR[GP1:90,2] + -13.229;
   1:L PR[91] R[100]mm/sec CNT100;
   1:  PR[GP1:91,1] = PR[GP1:90,1] + -1.408;
   1:  PR[GP1:91,2] = PR[GP1:90,2] + -12.499;
   1:L PR[91] R[100]mm/sec CNT100;
   1:  PR[GP1:91,1] = PR[GP1:90,1] + 1.681;
   1:  PR[GP1:91,2] = PR[GP1:90,2] + -12.469;
   1:L PR[91] R[100]mm/sec CNT100;
   1:  PR[GP1:91,1] = PR[GP1:90,1] + 3.314;
   1:  PR[GP1:91,2] = PR[GP1:90,2] + -14.426;
   1:L PR[91] R[100]mm/sec CNT100;
   1:  PR[GP1:91,1] = PR[GP1:90,1] + 4.279;
   1:  PR[GP1:91,2] = PR[GP1:90,2] + -15.034;
   1:L PR[91] R[100]mm/sec CNT100;
   1:  PR[GP1:91,1] = PR[GP1:90,1] + 4.705;
   1:  PR[GP1:91,2] = PR[GP1:90,2] + -15.267;
   1:L PR[91] R[100]mm/sec CNT100;
   1:  PR[GP1:91,1] = PR[GP1:90,1] + 7.787;
   1:  PR[GP1:91,2] = PR[GP1:90,2] + -19.484;
   1:L PR[91] R[100]mm/sec CNT100;
   1:  PR[GP1:91,1] = PR[GP1:90,1] + 10.598;
   1:  PR[GP1:91,2] = PR[GP1:90,2] + -23.560;
   1:L PR[91] R[100]mm/sec CNT100;
   1:  PR[GP1:91,1] = PR[GP1:90,1] + 11.379;
   1:  PR[GP1:91,2] = PR[GP1:90,2] + -24.316;
   1:L PR[91] R[100]mm/sec CNT100;
   1:  PR[GP1:91,1] = PR[GP1:90,1] + 18.423;
   1:  PR[GP1:91,2] = PR[GP1:90,2] + -29.761;
   1:L PR[91] R[100]mm/sec CNT100;
   1:  PR[GP1:91,1] = PR[GP1:90,1] + 21.639;
   1:  PR[GP1:91,2] = PR[GP1:90,2] + -31.329;
   1:L PR[91] R[100]mm/sec CNT100;
   1:  PR[GP1:91,1] = PR[GP1:90,1] + 27.852;
   1:  PR[GP1:91,2] = PR[GP1:90,2] + -33.688;
   1:L PR[91] R[100]mm/sec CNT100;
   1:  PR[GP1:91,1] = PR[GP1:90,1] + 34.008;
   1:  PR[GP1:91,2] = PR[GP1:90,2] + -34.594;
   1:L PR[91] R[100]mm/sec CNT100;
   1:  PR[GP1:91,1] = PR[GP1:90,1] + 38.255;
   1:  PR[GP1:91,2] = PR[GP1:90,2] + -34.897;
   1:L PR[91] R[100]mm/sec CNT100;
   1:  PR[GP1:91,1] = PR[GP1:90,1] + 46.773;
   1:  PR[GP1:91,2] = PR[GP1:90,2] + -33.525;
   1:L PR[91] R[100]mm/sec CNT100;
   1:  PR[GP1:91,1] = PR[GP1:90,1] + 48.794;
   1:  PR[GP1:91,2] = PR[GP1:90,2] + -33.072;
   1:L PR[91] R[100]mm/sec CNT100;
   1:  PR[GP1:91,1] = PR[GP1:90,1] + 58.194;
   1:  PR[GP1:91,2] = PR[GP1:90,2] + -28.353;
   1:L PR[91] R[100]mm/sec CNT100;
   1:  PR[GP1:91,1] = PR[GP1:90,1] + 58.477;
   1:  PR[GP1:91,2] = PR[GP1:90,2] + -28.193;
   1:L PR[91] R[100]mm/sec CNT100;
   1:  PR[GP1:91,1] = PR[GP1:90,1] + 66.242;
   1:  PR[GP1:91,2] = PR[GP1:90,2] + -20.549;
   1:L PR[91] R[100]mm/sec CNT100;
   1:  PR[GP1:91,1] = PR[GP1:90,1] + 66.554;
   1:  PR[GP1:91,2] = PR[GP1:90,2] + -19.979;
   1:L PR[91] R[100]mm/sec CNT100;
   1:  PR[GP1:91,1] = PR[GP1:90,1] + 71.264;
   1:  PR[GP1:91,2] = PR[GP1:90,2] + -10.890;
   1:L PR[91] R[100]mm/sec CNT100;
   1:  PR[GP1:91,1] = PR[GP1:90,1] + 71.487;
   1:  PR[GP1:91,2] = PR[GP1:90,2] + -9.573;
   1:L PR[91] R[100]mm/sec CNT100;
   1:  PR[GP1:91,1] = PR[GP1:90,1] + 73.007;
   1:  PR[GP1:91,2] = PR[GP1:90,2] + -0.075;
   1:L PR[91] R[100]mm/sec CNT100;
   1:  PR[GP1:91,1] = PR[GP1:90,1] + 72.752;
   1:  PR[GP1:91,2] = PR[GP1:90,2] + 1.434;
   1:L PR[91] R[100]mm/sec CNT100;
   1:  PR[GP1:91,1] = PR[GP1:90,1] + 71.263;
   1:  PR[GP1:91,2] = PR[GP1:90,2] + 10.748;
   1:L PR[91] R[100]mm/sec CNT100;
   1:  PR[GP1:91,1] = PR[GP1:90,1] + 66.554;
   1:  PR[GP1:91,2] = PR[GP1:90,2] + 19.835;
   1:L PR[91] R[100]mm/sec CNT100;
   1:  PR[GP1:91,1] = PR[GP1:90,1] + 66.242;
   1:  PR[GP1:91,2] = PR[GP1:90,2] + 20.405;
   1:L PR[91] R[100]mm/sec CNT100;
   1:  PR[GP1:91,1] = PR[GP1:90,1] + 58.477;
   1:  PR[GP1:91,2] = PR[GP1:90,2] + 28.049;
   1:L PR[91] R[100]mm/sec CNT100;
   1:  PR[GP1:91,1] = PR[GP1:90,1] + 58.194;
   1:  PR[GP1:91,2] = PR[GP1:90,2] + 28.209;
   1:L PR[91] R[100]mm/sec CNT100;
   1:  PR[GP1:91,1] = PR[GP1:90,1] + 48.794;
   1:  PR[GP1:91,2] = PR[GP1:90,2] + 32.928;
   1:L PR[91] R[100]mm/sec CNT100;
   1:  PR[GP1:91,1] = PR[GP1:90,1] + 46.773;
   1:  PR[GP1:91,2] = PR[GP1:90,2] + 33.381;
   1:L PR[91] R[100]mm/sec CNT100;
   1:  PR[GP1:91,1] = PR[GP1:90,1] + 38.255;
   1:  PR[GP1:91,2] = PR[GP1:90,2] + 34.753;
   1:L PR[91] R[100]mm/sec CNT100;
   1:  PR[GP1:91,1] = PR[GP1:90,1] + 34.008;
   1:  PR[GP1:91,2] = PR[GP1:90,2] + 34.450;
   1:L PR[91] R[100]mm/sec CNT100;
   1:  PR[GP1:91,1] = PR[GP1:90,1] + 27.852;
   1:  PR[GP1:91,2] = PR[GP1:90,2] + 33.544;
   1:L PR[91] R[100]mm/sec CNT100;
   1:  PR[GP1:91,1] = PR[GP1:90,1] + 21.639;
   1:  PR[GP1:91,2] = PR[GP1:90,2] + 31.185;
   1:L PR[91] R[100]mm/sec CNT100;
   1:  PR[GP1:91,1] = PR[GP1:90,1] + 18.423;
   1:  PR[GP1:91,2] = PR[GP1:90,2] + 29.617;
   1:L PR[91] R[100]mm/sec CNT100;
   1:  PR[GP1:91,1] = PR[GP1:90,1] + 11.379;
   1:  PR[GP1:91,2] = PR[GP1:90,2] + 24.172;
   1:L PR[91] R[100]mm/sec CNT100;
   1:  PR[GP1:91,1] = PR[GP1:90,1] + 10.598;
   1:  PR[GP1:91,2] = PR[GP1:90,2] + 23.416;
   1:L PR[91] R[100]mm/sec CNT100;
   1:  PR[GP1:91,1] = PR[GP1:90,1] + 7.730;
   1:  PR[GP1:91,2] = PR[GP1:90,2] + 19.262;
   1:L PR[91] R[100]mm/sec CNT100;
   1:  PR[GP1:91,1] = PR[GP1:90,1] + 4.765;
   1:  PR[GP1:91,2] = PR[GP1:90,2] + 15.206;
   1:L PR[91] R[100]mm/sec CNT100;
   1:  PR[GP1:91,1] = PR[GP1:90,1] + 2.811;
   1:  PR[GP1:91,2] = PR[GP1:90,2] + 13.055;
   1:L PR[91] R[100]mm/sec CNT100;
   1:  PR[GP1:91,1] = PR[GP1:90,1] + 1.562;
   1:  PR[GP1:91,2] = PR[GP1:90,2] + 12.326;
   1:L PR[91] R[100]mm/sec CNT100;
   1:  PR[GP1:91,1] = PR[GP1:90,1] + -1.408;
   1:  PR[GP1:91,2] = PR[GP1:90,2] + 12.355;
   1:L PR[91] R[100]mm/sec CNT100;
   1:  ! -- Layer/Ebene 50 -- !;
   1:  PR[91] = PR[90];
   1:  PR[GP1:91,1] = PR[GP1:90,1] + -2.774;
   1:  PR[GP1:91,2] = PR[GP1:90,2] + 13.636;
   1:  PR[GP1:91,3] = PR[GP1:90,3] + 30.805;
   1:L PR[91] R[100]mm/sec CNT100;
   1:  PR[GP1:91,1] = PR[GP1:90,1] + -4.619;
   1:  PR[GP1:91,2] = PR[GP1:90,2] + 15.626;
   1:L PR[91] R[100]mm/sec CNT100;
   1:  PR[GP1:91,1] = PR[GP1:90,1] + -4.632;
   1:  PR[GP1:91,2] = PR[GP1:90,2] + 15.746;
   1:L PR[91] R[100]mm/sec CNT100;
   1:  PR[GP1:91,1] = PR[GP1:90,1] + -9.941;
   1:  PR[GP1:91,2] = PR[GP1:90,2] + 23.006;
   1:L PR[91] R[100]mm/sec CNT100;
   1:  PR[GP1:91,1] = PR[GP1:90,1] + -10.430;
   1:  PR[GP1:91,2] = PR[GP1:90,2] + 23.714;
   1:L PR[91] R[100]mm/sec CNT100;
   1:  PR[GP1:91,1] = PR[GP1:90,1] + -10.514;
   1:  PR[GP1:91,2] = PR[GP1:90,2] + 23.795;
   1:L PR[91] R[100]mm/sec CNT100;
   1:  PR[GP1:91,1] = PR[GP1:90,1] + -18.287;
   1:  PR[GP1:91,2] = PR[GP1:90,2] + 29.796;
   1:L PR[91] R[100]mm/sec CNT100;
   1:  PR[GP1:91,1] = PR[GP1:90,1] + -20.670;
   1:  PR[GP1:91,2] = PR[GP1:90,2] + 30.959;
   1:L PR[91] R[100]mm/sec CNT100;
   1:  PR[GP1:91,1] = PR[GP1:90,1] + -27.710;
   1:  PR[GP1:91,2] = PR[GP1:90,2] + 33.635;
   1:L PR[91] R[100]mm/sec CNT100;
   1:  PR[GP1:91,1] = PR[GP1:90,1] + -33.003;
   1:  PR[GP1:91,2] = PR[GP1:90,2] + 34.411;
   1:L PR[91] R[100]mm/sec CNT100;
   1:  PR[GP1:91,1] = PR[GP1:90,1] + -38.083;
   1:  PR[GP1:91,2] = PR[GP1:90,2] + 34.773;
   1:L PR[91] R[100]mm/sec CNT100;
   1:  PR[GP1:91,1] = PR[GP1:90,1] + -45.800;
   1:  PR[GP1:91,2] = PR[GP1:90,2] + 33.529;
   1:L PR[91] R[100]mm/sec CNT100;
   1:  PR[GP1:91,1] = PR[GP1:90,1] + -48.581;
   1:  PR[GP1:91,2] = PR[GP1:90,2] + 32.907;
   1:L PR[91] R[100]mm/sec CNT100;
   1:  PR[GP1:91,1] = PR[GP1:90,1] + -57.309;
   1:  PR[GP1:91,2] = PR[GP1:90,2] + 28.517;
   1:L PR[91] R[100]mm/sec CNT100;
   1:  PR[GP1:91,1] = PR[GP1:90,1] + -58.220;
   1:  PR[GP1:91,2] = PR[GP1:90,2] + 28.003;
   1:L PR[91] R[100]mm/sec CNT100;
   1:  PR[GP1:91,1] = PR[GP1:90,1] + -65.996;
   1:  PR[GP1:91,2] = PR[GP1:90,2] + 20.372;
   1:L PR[91] R[100]mm/sec CNT100;
   1:  PR[GP1:91,1] = PR[GP1:90,1] + -70.994;
   1:  PR[GP1:91,2] = PR[GP1:90,2] + 10.706;
   1:L PR[91] R[100]mm/sec CNT100;
   1:  PR[GP1:91,1] = PR[GP1:90,1] + -72.728;
   1:  PR[GP1:91,2] = PR[GP1:90,2] + -0.069;
   1:L PR[91] R[100]mm/sec CNT100;
   1:  PR[GP1:91,1] = PR[GP1:90,1] + -72.571;
   1:  PR[GP1:91,2] = PR[GP1:90,2] + -0.992;
   1:L PR[91] R[100]mm/sec CNT100;
   1:  PR[GP1:91,1] = PR[GP1:90,1] + -70.993;
   1:  PR[GP1:91,2] = PR[GP1:90,2] + -10.851;
   1:L PR[91] R[100]mm/sec CNT100;
   1:  PR[GP1:91,1] = PR[GP1:90,1] + -65.996;
   1:  PR[GP1:91,2] = PR[GP1:90,2] + -20.516;
   1:L PR[91] R[100]mm/sec CNT100;
   1:  PR[GP1:91,1] = PR[GP1:90,1] + -58.220;
   1:  PR[GP1:91,2] = PR[GP1:90,2] + -28.147;
   1:L PR[91] R[100]mm/sec CNT100;
   1:  PR[GP1:91,1] = PR[GP1:90,1] + -57.309;
   1:  PR[GP1:91,2] = PR[GP1:90,2] + -28.661;
   1:L PR[91] R[100]mm/sec CNT100;
   1:  PR[GP1:91,1] = PR[GP1:90,1] + -48.581;
   1:  PR[GP1:91,2] = PR[GP1:90,2] + -33.050;
   1:L PR[91] R[100]mm/sec CNT100;
   1:  PR[GP1:91,1] = PR[GP1:90,1] + -45.800;
   1:  PR[GP1:91,2] = PR[GP1:90,2] + -33.673;
   1:L PR[91] R[100]mm/sec CNT100;
   1:  PR[GP1:91,1] = PR[GP1:90,1] + -38.084;
   1:  PR[GP1:91,2] = PR[GP1:90,2] + -34.916;
   1:L PR[91] R[100]mm/sec CNT100;
   1:  PR[GP1:91,1] = PR[GP1:90,1] + -33.003;
   1:  PR[GP1:91,2] = PR[GP1:90,2] + -34.555;
   1:L PR[91] R[100]mm/sec CNT100;
   1:  PR[GP1:91,1] = PR[GP1:90,1] + -27.710;
   1:  PR[GP1:91,2] = PR[GP1:90,2] + -33.779;
   1:L PR[91] R[100]mm/sec CNT100;
   1:  PR[GP1:91,1] = PR[GP1:90,1] + -20.670;
   1:  PR[GP1:91,2] = PR[GP1:90,2] + -31.103;
   1:L PR[91] R[100]mm/sec CNT100;
   1:  PR[GP1:91,1] = PR[GP1:90,1] + -18.287;
   1:  PR[GP1:91,2] = PR[GP1:90,2] + -29.940;
   1:L PR[91] R[100]mm/sec CNT100;
   1:  PR[GP1:91,1] = PR[GP1:90,1] + -10.514;
   1:  PR[GP1:91,2] = PR[GP1:90,2] + -23.939;
   1:L PR[91] R[100]mm/sec CNT100;
   1:  PR[GP1:91,1] = PR[GP1:90,1] + -10.430;
   1:  PR[GP1:91,2] = PR[GP1:90,2] + -23.858;
   1:L PR[91] R[100]mm/sec CNT100;
   1:  PR[GP1:91,1] = PR[GP1:90,1] + -9.951;
   1:  PR[GP1:91,2] = PR[GP1:90,2] + -23.164;
   1:L PR[91] R[100]mm/sec CNT100;
   1:  PR[GP1:91,1] = PR[GP1:90,1] + -4.521;
   1:  PR[GP1:91,2] = PR[GP1:90,2] + -15.738;
   1:L PR[91] R[100]mm/sec CNT100;
   1:  PR[GP1:91,1] = PR[GP1:90,1] + -2.779;
   1:  PR[GP1:91,2] = PR[GP1:90,2] + -13.783;
   1:L PR[91] R[100]mm/sec CNT100;
   1:  PR[GP1:91,1] = PR[GP1:90,1] + -1.305;
   1:  PR[GP1:91,2] = PR[GP1:90,2] + -12.921;
   1:L PR[91] R[100]mm/sec CNT100;
   1:  PR[GP1:91,1] = PR[GP1:90,1] + 1.582;
   1:  PR[GP1:91,2] = PR[GP1:90,2] + -12.893;
   1:L PR[91] R[100]mm/sec CNT100;
   1:  PR[GP1:91,1] = PR[GP1:90,1] + 3.100;
   1:  PR[GP1:91,2] = PR[GP1:90,2] + -14.711;
   1:L PR[91] R[100]mm/sec CNT100;
   1:  PR[GP1:91,1] = PR[GP1:90,1] + 3.984;
   1:  PR[GP1:91,2] = PR[GP1:90,2] + -15.268;
   1:L PR[91] R[100]mm/sec CNT100;
   1:  PR[GP1:91,1] = PR[GP1:90,1] + 4.671;
   1:  PR[GP1:91,2] = PR[GP1:90,2] + -15.644;
   1:L PR[91] R[100]mm/sec CNT100;
   1:  PR[GP1:91,1] = PR[GP1:90,1] + 10.166;
   1:  PR[GP1:91,2] = PR[GP1:90,2] + -23.162;
   1:L PR[91] R[100]mm/sec CNT100;
   1:  PR[GP1:91,1] = PR[GP1:90,1] + 10.643;
   1:  PR[GP1:91,2] = PR[GP1:90,2] + -23.854;
   1:L PR[91] R[100]mm/sec CNT100;
   1:  PR[GP1:91,1] = PR[GP1:90,1] + 10.727;
   1:  PR[GP1:91,2] = PR[GP1:90,2] + -23.936;
   1:L PR[91] R[100]mm/sec CNT100;
   1:  PR[GP1:91,1] = PR[GP1:90,1] + 18.498;
   1:  PR[GP1:91,2] = PR[GP1:90,2] + -29.942;
   1:L PR[91] R[100]mm/sec CNT100;
   1:  PR[GP1:91,1] = PR[GP1:90,1] + 20.879;
   1:  PR[GP1:91,2] = PR[GP1:90,2] + -31.104;
   1:L PR[91] R[100]mm/sec CNT100;
   1:  PR[GP1:91,1] = PR[GP1:90,1] + 27.918;
   1:  PR[GP1:91,2] = PR[GP1:90,2] + -33.775;
   1:L PR[91] R[100]mm/sec CNT100;
   1:  PR[GP1:91,1] = PR[GP1:90,1] + 33.210;
   1:  PR[GP1:91,2] = PR[GP1:90,2] + -34.555;
   1:L PR[91] R[100]mm/sec CNT100;
   1:  PR[GP1:91,1] = PR[GP1:90,1] + 38.290;
   1:  PR[GP1:91,2] = PR[GP1:90,2] + -34.917;
   1:L PR[91] R[100]mm/sec CNT100;
   1:  PR[GP1:91,1] = PR[GP1:90,1] + 46.005;
   1:  PR[GP1:91,2] = PR[GP1:90,2] + -33.674;
   1:L PR[91] R[100]mm/sec CNT100;
   1:  PR[GP1:91,1] = PR[GP1:90,1] + 48.787;
   1:  PR[GP1:91,2] = PR[GP1:90,2] + -33.050;
   1:L PR[91] R[100]mm/sec CNT100;
   1:  PR[GP1:91,1] = PR[GP1:90,1] + 57.516;
   1:  PR[GP1:91,2] = PR[GP1:90,2] + -28.668;
   1:L PR[91] R[100]mm/sec CNT100;
   1:  PR[GP1:91,1] = PR[GP1:90,1] + 58.428;
   1:  PR[GP1:91,2] = PR[GP1:90,2] + -28.155;
   1:L PR[91] R[100]mm/sec CNT100;
   1:  PR[GP1:91,1] = PR[GP1:90,1] + 66.207;
   1:  PR[GP1:91,2] = PR[GP1:90,2] + -20.510;
   1:L PR[91] R[100]mm/sec CNT100;
   1:  PR[GP1:91,1] = PR[GP1:90,1] + 71.206;
   1:  PR[GP1:91,2] = PR[GP1:90,2] + -10.867;
   1:L PR[91] R[100]mm/sec CNT100;
   1:  PR[GP1:91,1] = PR[GP1:90,1] + 72.941;
   1:  PR[GP1:91,2] = PR[GP1:90,2] + -0.072;
   1:L PR[91] R[100]mm/sec CNT100;
   1:  PR[GP1:91,1] = PR[GP1:90,1] + 71.206;
   1:  PR[GP1:91,2] = PR[GP1:90,2] + 10.723;
   1:L PR[91] R[100]mm/sec CNT100;
   1:  PR[GP1:91,1] = PR[GP1:90,1] + 66.206;
   1:  PR[GP1:91,2] = PR[GP1:90,2] + 20.366;
   1:L PR[91] R[100]mm/sec CNT100;
   1:  PR[GP1:91,1] = PR[GP1:90,1] + 58.428;
   1:  PR[GP1:91,2] = PR[GP1:90,2] + 28.011;
   1:L PR[91] R[100]mm/sec CNT100;
   1:  PR[GP1:91,1] = PR[GP1:90,1] + 57.516;
   1:  PR[GP1:91,2] = PR[GP1:90,2] + 28.524;
   1:L PR[91] R[100]mm/sec CNT100;
   1:  PR[GP1:91,1] = PR[GP1:90,1] + 48.787;
   1:  PR[GP1:91,2] = PR[GP1:90,2] + 32.906;
   1:L PR[91] R[100]mm/sec CNT100;
   1:  PR[GP1:91,1] = PR[GP1:90,1] + 46.005;
   1:  PR[GP1:91,2] = PR[GP1:90,2] + 33.530;
   1:L PR[91] R[100]mm/sec CNT100;
   1:  PR[GP1:91,1] = PR[GP1:90,1] + 38.290;
   1:  PR[GP1:91,2] = PR[GP1:90,2] + 34.773;
   1:L PR[91] R[100]mm/sec CNT100;
   1:  PR[GP1:91,1] = PR[GP1:90,1] + 33.210;
   1:  PR[GP1:91,2] = PR[GP1:90,2] + 34.411;
   1:L PR[91] R[100]mm/sec CNT100;
   1:  PR[GP1:91,1] = PR[GP1:90,1] + 27.918;
   1:  PR[GP1:91,2] = PR[GP1:90,2] + 33.631;
   1:L PR[91] R[100]mm/sec CNT100;
   1:  PR[GP1:91,1] = PR[GP1:90,1] + 20.879;
   1:  PR[GP1:91,2] = PR[GP1:90,2] + 30.960;
   1:L PR[91] R[100]mm/sec CNT100;
   1:  PR[GP1:91,1] = PR[GP1:90,1] + 18.498;
   1:  PR[GP1:91,2] = PR[GP1:90,2] + 29.798;
   1:L PR[91] R[100]mm/sec CNT100;
   1:  PR[GP1:91,1] = PR[GP1:90,1] + 10.728;
   1:  PR[GP1:91,2] = PR[GP1:90,2] + 23.792;
   1:L PR[91] R[100]mm/sec CNT100;
   1:  PR[GP1:91,1] = PR[GP1:90,1] + 10.643;
   1:  PR[GP1:91,2] = PR[GP1:90,2] + 23.710;
   1:L PR[91] R[100]mm/sec CNT100;
   1:  PR[GP1:91,1] = PR[GP1:90,1] + 10.155;
   1:  PR[GP1:91,2] = PR[GP1:90,2] + 23.004;
   1:L PR[91] R[100]mm/sec CNT100;
   1:  PR[GP1:91,1] = PR[GP1:90,1] + 4.731;
   1:  PR[GP1:91,2] = PR[GP1:90,2] + 15.583;
   1:L PR[91] R[100]mm/sec CNT100;
   1:  PR[GP1:91,1] = PR[GP1:90,1] + 2.939;
   1:  PR[GP1:91,2] = PR[GP1:90,2] + 13.611;
   1:L PR[91] R[100]mm/sec CNT100;
   1:  PR[GP1:91,1] = PR[GP1:90,1] + 1.463;
   1:  PR[GP1:91,2] = PR[GP1:90,2] + 12.750;
   1:L PR[91] R[100]mm/sec CNT100;
   1:  PR[GP1:91,1] = PR[GP1:90,1] + -1.305;
   1:  PR[GP1:91,2] = PR[GP1:90,2] + 12.777;
   1:L PR[91] R[100]mm/sec CNT100;
   1:  ! -- Layer/Ebene 51 -- !;
   1:  PR[91] = PR[90];
   1:  PR[GP1:91,1] = PR[GP1:90,1] + -2.897;
   1:  PR[GP1:91,2] = PR[GP1:90,2] + 14.190;
   1:  PR[GP1:91,3] = PR[GP1:90,3] + 31.415;
   1:L PR[91] R[100]mm/sec CNT100;
   1:  PR[GP1:91,1] = PR[GP1:90,1] + -4.584;
   1:  PR[GP1:91,2] = PR[GP1:90,2] + 16.011;
   1:L PR[91] R[100]mm/sec CNT100;
   1:  PR[GP1:91,1] = PR[GP1:90,1] + -4.597;
   1:  PR[GP1:91,2] = PR[GP1:90,2] + 16.123;
   1:L PR[91] R[100]mm/sec CNT100;
   1:  PR[GP1:91,1] = PR[GP1:90,1] + -9.970;
   1:  PR[GP1:91,2] = PR[GP1:90,2] + 23.471;
   1:L PR[91] R[100]mm/sec CNT100;
   1:  PR[GP1:91,1] = PR[GP1:90,1] + -10.239;
   1:  PR[GP1:91,2] = PR[GP1:90,2] + 23.785;
   1:L PR[91] R[100]mm/sec CNT100;
   1:  PR[GP1:91,1] = PR[GP1:90,1] + -12.689;
   1:  PR[GP1:91,2] = PR[GP1:90,2] + 25.598;
   1:L PR[91] R[100]mm/sec CNT100;
   1:  PR[GP1:91,1] = PR[GP1:90,1] + -18.360;
   1:  PR[GP1:91,2] = PR[GP1:90,2] + 29.976;
   1:L PR[91] R[100]mm/sec CNT100;
   1:  PR[GP1:91,1] = PR[GP1:90,1] + -19.910;
   1:  PR[GP1:91,2] = PR[GP1:90,2] + 30.732;
   1:L PR[91] R[100]mm/sec CNT100;
   1:  PR[GP1:91,1] = PR[GP1:90,1] + -27.775;
   1:  PR[GP1:91,2] = PR[GP1:90,2] + 33.722;
   1:L PR[91] R[100]mm/sec CNT100;
   1:  PR[GP1:91,1] = PR[GP1:90,1] + -32.203;
   1:  PR[GP1:91,2] = PR[GP1:90,2] + 34.372;
   1:L PR[91] R[100]mm/sec CNT100;
   1:  PR[GP1:91,1] = PR[GP1:90,1] + -38.118;
   1:  PR[GP1:91,2] = PR[GP1:90,2] + 34.792;
   1:L PR[91] R[100]mm/sec CNT100;
   1:  PR[GP1:91,1] = PR[GP1:90,1] + -45.031;
   1:  PR[GP1:91,2] = PR[GP1:90,2] + 33.678;
   1:L PR[91] R[100]mm/sec CNT100;
   1:  PR[GP1:91,1] = PR[GP1:90,1] + -48.573;
   1:  PR[GP1:91,2] = PR[GP1:90,2] + 32.885;
   1:L PR[91] R[100]mm/sec CNT100;
   1:  PR[GP1:91,1] = PR[GP1:90,1] + -56.631;
   1:  PR[GP1:91,2] = PR[GP1:90,2] + 28.833;
   1:L PR[91] R[100]mm/sec CNT100;
   1:  PR[GP1:91,1] = PR[GP1:90,1] + -58.170;
   1:  PR[GP1:91,2] = PR[GP1:90,2] + 27.965;
   1:L PR[91] R[100]mm/sec CNT100;
   1:  PR[GP1:91,1] = PR[GP1:90,1] + -65.594;
   1:  PR[GP1:91,2] = PR[GP1:90,2] + 20.681;
   1:L PR[91] R[100]mm/sec CNT100;
   1:  PR[GP1:91,1] = PR[GP1:90,1] + -65.915;
   1:  PR[GP1:91,2] = PR[GP1:90,2] + 20.343;
   1:L PR[91] R[100]mm/sec CNT100;
   1:  PR[GP1:91,1] = PR[GP1:90,1] + -70.938;
   1:  PR[GP1:91,2] = PR[GP1:90,2] + 10.678;
   1:L PR[91] R[100]mm/sec CNT100;
   1:  PR[GP1:91,1] = PR[GP1:90,1] + -70.950;
   1:  PR[GP1:91,2] = PR[GP1:90,2] + 10.605;
   1:L PR[91] R[100]mm/sec CNT100;
   1:  PR[GP1:91,1] = PR[GP1:90,1] + -72.662;
   1:  PR[GP1:91,2] = PR[GP1:90,2] + -0.072;
   1:L PR[91] R[100]mm/sec CNT100;
   1:  PR[GP1:91,1] = PR[GP1:90,1] + -70.937;
   1:  PR[GP1:91,2] = PR[GP1:90,2] + -10.825;
   1:L PR[91] R[100]mm/sec CNT100;
   1:  PR[GP1:91,1] = PR[GP1:90,1] + -69.746;
   1:  PR[GP1:91,2] = PR[GP1:90,2] + -13.130;
   1:L PR[91] R[100]mm/sec CNT100;
   1:  PR[GP1:91,1] = PR[GP1:90,1] + -65.915;
   1:  PR[GP1:91,2] = PR[GP1:90,2] + -20.487;
   1:L PR[91] R[100]mm/sec CNT100;
   1:  PR[GP1:91,1] = PR[GP1:90,1] + -65.594;
   1:  PR[GP1:91,2] = PR[GP1:90,2] + -20.825;
   1:L PR[91] R[100]mm/sec CNT100;
   1:  PR[GP1:91,1] = PR[GP1:90,1] + -58.170;
   1:  PR[GP1:91,2] = PR[GP1:90,2] + -28.109;
   1:L PR[91] R[100]mm/sec CNT100;
   1:  PR[GP1:91,1] = PR[GP1:90,1] + -56.631;
   1:  PR[GP1:91,2] = PR[GP1:90,2] + -28.976;
   1:L PR[91] R[100]mm/sec CNT100;
   1:  PR[GP1:91,1] = PR[GP1:90,1] + -48.573;
   1:  PR[GP1:91,2] = PR[GP1:90,2] + -33.029;
   1:L PR[91] R[100]mm/sec CNT100;
   1:  PR[GP1:91,1] = PR[GP1:90,1] + -45.031;
   1:  PR[GP1:91,2] = PR[GP1:90,2] + -33.822;
   1:L PR[91] R[100]mm/sec CNT100;
   1:  PR[GP1:91,1] = PR[GP1:90,1] + -38.118;
   1:  PR[GP1:91,2] = PR[GP1:90,2] + -34.936;
   1:L PR[91] R[100]mm/sec CNT100;
   1:  PR[GP1:91,1] = PR[GP1:90,1] + -32.203;
   1:  PR[GP1:91,2] = PR[GP1:90,2] + -34.515;
   1:L PR[91] R[100]mm/sec CNT100;
   1:  PR[GP1:91,1] = PR[GP1:90,1] + -27.775;
   1:  PR[GP1:91,2] = PR[GP1:90,2] + -33.866;
   1:L PR[91] R[100]mm/sec CNT100;
   1:  PR[GP1:91,1] = PR[GP1:90,1] + -19.910;
   1:  PR[GP1:91,2] = PR[GP1:90,2] + -30.876;
   1:L PR[91] R[100]mm/sec CNT100;
   1:  PR[GP1:91,1] = PR[GP1:90,1] + -18.360;
   1:  PR[GP1:91,2] = PR[GP1:90,2] + -30.120;
   1:L PR[91] R[100]mm/sec CNT100;
   1:  PR[GP1:91,1] = PR[GP1:90,1] + -12.688;
   1:  PR[GP1:91,2] = PR[GP1:90,2] + -25.741;
   1:L PR[91] R[100]mm/sec CNT100;
   1:  PR[GP1:91,1] = PR[GP1:90,1] + -10.479;
   1:  PR[GP1:91,2] = PR[GP1:90,2] + -24.123;
   1:L PR[91] R[100]mm/sec CNT100;
   1:  PR[GP1:91,1] = PR[GP1:90,1] + -10.246;
   1:  PR[GP1:91,2] = PR[GP1:90,2] + -23.937;
   1:L PR[91] R[100]mm/sec CNT100;
   1:  PR[GP1:91,1] = PR[GP1:90,1] + -9.970;
   1:  PR[GP1:91,2] = PR[GP1:90,2] + -23.615;
   1:L PR[91] R[100]mm/sec CNT100;
   1:  PR[GP1:91,1] = PR[GP1:90,1] + -4.485;
   1:  PR[GP1:91,2] = PR[GP1:90,2] + -16.114;
   1:L PR[91] R[100]mm/sec CNT100;
   1:  PR[GP1:91,1] = PR[GP1:90,1] + -2.902;
   1:  PR[GP1:91,2] = PR[GP1:90,2] + -14.337;
   1:L PR[91] R[100]mm/sec CNT100;
   1:  PR[GP1:91,1] = PR[GP1:90,1] + -1.201;
   1:  PR[GP1:91,2] = PR[GP1:90,2] + -13.343;
   1:L PR[91] R[100]mm/sec CNT100;
   1:  PR[GP1:91,1] = PR[GP1:90,1] + 1.484;
   1:  PR[GP1:91,2] = PR[GP1:90,2] + -13.316;
   1:L PR[91] R[100]mm/sec CNT100;
   1:  PR[GP1:91,1] = PR[GP1:90,1] + 2.886;
   1:  PR[GP1:91,2] = PR[GP1:90,2] + -14.997;
   1:L PR[91] R[100]mm/sec CNT100;
   1:  PR[GP1:91,1] = PR[GP1:90,1] + 3.689;
   1:  PR[GP1:91,2] = PR[GP1:90,2] + -15.503;
   1:L PR[91] R[100]mm/sec CNT100;
   1:  PR[GP1:91,1] = PR[GP1:90,1] + 4.637;
   1:  PR[GP1:91,2] = PR[GP1:90,2] + -16.022;
   1:L PR[91] R[100]mm/sec CNT100;
   1:  PR[GP1:91,1] = PR[GP1:90,1] + 10.185;
   1:  PR[GP1:91,2] = PR[GP1:90,2] + -23.612;
   1:L PR[91] R[100]mm/sec CNT100;
   1:  PR[GP1:91,1] = PR[GP1:90,1] + 10.455;
   1:  PR[GP1:91,2] = PR[GP1:90,2] + -23.929;
   1:L PR[91] R[100]mm/sec CNT100;
   1:  PR[GP1:91,1] = PR[GP1:90,1] + 12.903;
   1:  PR[GP1:91,2] = PR[GP1:90,2] + -25.740;
   1:L PR[91] R[100]mm/sec CNT100;
   1:  PR[GP1:91,1] = PR[GP1:90,1] + 18.572;
   1:  PR[GP1:91,2] = PR[GP1:90,2] + -30.123;
   1:L PR[91] R[100]mm/sec CNT100;
   1:  PR[GP1:91,1] = PR[GP1:90,1] + 20.120;
   1:  PR[GP1:91,2] = PR[GP1:90,2] + -30.878;
   1:L PR[91] R[100]mm/sec CNT100;
   1:  PR[GP1:91,1] = PR[GP1:90,1] + 27.984;
   1:  PR[GP1:91,2] = PR[GP1:90,2] + -33.863;
   1:L PR[91] R[100]mm/sec CNT100;
   1:  PR[GP1:91,1] = PR[GP1:90,1] + 32.411;
   1:  PR[GP1:91,2] = PR[GP1:90,2] + -34.515;
   1:L PR[91] R[100]mm/sec CNT100;
   1:  PR[GP1:91,1] = PR[GP1:90,1] + 38.325;
   1:  PR[GP1:91,2] = PR[GP1:90,2] + -34.937;
   1:L PR[91] R[100]mm/sec CNT100;
   1:  PR[GP1:91,1] = PR[GP1:90,1] + 45.238;
   1:  PR[GP1:91,2] = PR[GP1:90,2] + -33.823;
   1:L PR[91] R[100]mm/sec CNT100;
   1:  PR[GP1:91,1] = PR[GP1:90,1] + 48.780;
   1:  PR[GP1:91,2] = PR[GP1:90,2] + -33.029;
   1:L PR[91] R[100]mm/sec CNT100;
   1:  PR[GP1:91,1] = PR[GP1:90,1] + 56.839;
   1:  PR[GP1:91,2] = PR[GP1:90,2] + -28.982;
   1:L PR[91] R[100]mm/sec CNT100;
   1:  PR[GP1:91,1] = PR[GP1:90,1] + 58.378;
   1:  PR[GP1:91,2] = PR[GP1:90,2] + -28.116;
   1:L PR[91] R[100]mm/sec CNT100;
   1:  PR[GP1:91,1] = PR[GP1:90,1] + 65.804;
   1:  PR[GP1:91,2] = PR[GP1:90,2] + -20.821;
   1:L PR[91] R[100]mm/sec CNT100;
   1:  PR[GP1:91,1] = PR[GP1:90,1] + 66.125;
   1:  PR[GP1:91,2] = PR[GP1:90,2] + -20.481;
   1:L PR[91] R[100]mm/sec CNT100;
   1:  PR[GP1:91,1] = PR[GP1:90,1] + 71.149;
   1:  PR[GP1:91,2] = PR[GP1:90,2] + -10.842;
   1:L PR[91] R[100]mm/sec CNT100;
   1:  PR[GP1:91,1] = PR[GP1:90,1] + 72.875;
   1:  PR[GP1:91,2] = PR[GP1:90,2] + -0.072;
   1:L PR[91] R[100]mm/sec CNT100;
   1:  PR[GP1:91,1] = PR[GP1:90,1] + 71.149;
   1:  PR[GP1:91,2] = PR[GP1:90,2] + 10.698;
   1:L PR[91] R[100]mm/sec CNT100;
   1:  PR[GP1:91,1] = PR[GP1:90,1] + 66.125;
   1:  PR[GP1:91,2] = PR[GP1:90,2] + 20.337;
   1:L PR[91] R[100]mm/sec CNT100;
   1:  PR[GP1:91,1] = PR[GP1:90,1] + 65.804;
   1:  PR[GP1:91,2] = PR[GP1:90,2] + 20.677;
   1:L PR[91] R[100]mm/sec CNT100;
   1:  PR[GP1:91,1] = PR[GP1:90,1] + 58.378;
   1:  PR[GP1:91,2] = PR[GP1:90,2] + 27.972;
   1:L PR[91] R[100]mm/sec CNT100;
   1:  PR[GP1:91,1] = PR[GP1:90,1] + 56.839;
   1:  PR[GP1:91,2] = PR[GP1:90,2] + 28.838;
   1:L PR[91] R[100]mm/sec CNT100;
   1:  PR[GP1:91,1] = PR[GP1:90,1] + 48.780;
   1:  PR[GP1:91,2] = PR[GP1:90,2] + 32.885;
   1:L PR[91] R[100]mm/sec CNT100;
   1:  PR[GP1:91,1] = PR[GP1:90,1] + 45.238;
   1:  PR[GP1:91,2] = PR[GP1:90,2] + 33.679;
   1:L PR[91] R[100]mm/sec CNT100;
   1:  PR[GP1:91,1] = PR[GP1:90,1] + 38.325;
   1:  PR[GP1:91,2] = PR[GP1:90,2] + 34.793;
   1:L PR[91] R[100]mm/sec CNT100;
   1:  PR[GP1:91,1] = PR[GP1:90,1] + 32.411;
   1:  PR[GP1:91,2] = PR[GP1:90,2] + 34.371;
   1:L PR[91] R[100]mm/sec CNT100;
   1:  PR[GP1:91,1] = PR[GP1:90,1] + 27.984;
   1:  PR[GP1:91,2] = PR[GP1:90,2] + 33.719;
   1:L PR[91] R[100]mm/sec CNT100;
   1:  PR[GP1:91,1] = PR[GP1:90,1] + 20.120;
   1:  PR[GP1:91,2] = PR[GP1:90,2] + 30.734;
   1:L PR[91] R[100]mm/sec CNT100;
   1:  PR[GP1:91,1] = PR[GP1:90,1] + 18.572;
   1:  PR[GP1:91,2] = PR[GP1:90,2] + 29.979;
   1:L PR[91] R[100]mm/sec CNT100;
   1:  PR[GP1:91,1] = PR[GP1:90,1] + 12.901;
   1:  PR[GP1:91,2] = PR[GP1:90,2] + 25.595;
   1:L PR[91] R[100]mm/sec CNT100;
   1:  PR[GP1:91,1] = PR[GP1:90,1] + 10.693;
   1:  PR[GP1:91,2] = PR[GP1:90,2] + 23.977;
   1:L PR[91] R[100]mm/sec CNT100;
   1:  PR[GP1:91,1] = PR[GP1:90,1] + 10.462;
   1:  PR[GP1:91,2] = PR[GP1:90,2] + 23.793;
   1:L PR[91] R[100]mm/sec CNT100;
   1:  PR[GP1:91,1] = PR[GP1:90,1] + 10.185;
   1:  PR[GP1:91,2] = PR[GP1:90,2] + 23.468;
   1:L PR[91] R[100]mm/sec CNT100;
   1:  PR[GP1:91,1] = PR[GP1:90,1] + 4.697;
   1:  PR[GP1:91,2] = PR[GP1:90,2] + 15.961;
   1:L PR[91] R[100]mm/sec CNT100;
   1:  PR[GP1:91,1] = PR[GP1:90,1] + 3.068;
   1:  PR[GP1:91,2] = PR[GP1:90,2] + 14.167;
   1:L PR[91] R[100]mm/sec CNT100;
   1:  PR[GP1:91,1] = PR[GP1:90,1] + 1.365;
   1:  PR[GP1:91,2] = PR[GP1:90,2] + 13.174;
   1:L PR[91] R[100]mm/sec CNT100;
   1:  PR[GP1:91,1] = PR[GP1:90,1] + -1.201;
   1:  PR[GP1:91,2] = PR[GP1:90,2] + 13.199;
   1:L PR[91] R[100]mm/sec CNT100;
   1:  ! -- Layer/Ebene 52 -- !;
   1:  PR[91] = PR[90];
   1:  PR[GP1:91,1] = PR[GP1:90,1] + -3.019;
   1:  PR[GP1:91,2] = PR[GP1:90,2] + 14.744;
   1:  PR[GP1:91,3] = PR[GP1:90,3] + 32.025;
   1:L PR[91] R[100]mm/sec CNT100;
   1:  PR[GP1:91,1] = PR[GP1:90,1] + -4.549;
   1:  PR[GP1:91,2] = PR[GP1:90,2] + 16.395;
   1:L PR[91] R[100]mm/sec CNT100;
   1:  PR[GP1:91,1] = PR[GP1:90,1] + -4.561;
   1:  PR[GP1:91,2] = PR[GP1:90,2] + 16.500;
   1:L PR[91] R[100]mm/sec CNT100;
   1:  PR[GP1:91,1] = PR[GP1:90,1] + -9.357;
   1:  PR[GP1:91,2] = PR[GP1:90,2] + 23.058;
   1:L PR[91] R[100]mm/sec CNT100;
   1:  PR[GP1:91,1] = PR[GP1:90,1] + -10.044;
   1:  PR[GP1:91,2] = PR[GP1:90,2] + 23.861;
   1:L PR[91] R[100]mm/sec CNT100;
   1:  PR[GP1:91,1] = PR[GP1:90,1] + -15.688;
   1:  PR[GP1:91,2] = PR[GP1:90,2] + 28.036;
   1:L PR[91] R[100]mm/sec CNT100;
   1:  PR[GP1:91,1] = PR[GP1:90,1] + -18.434;
   1:  PR[GP1:91,2] = PR[GP1:90,2] + 30.156;
   1:L PR[91] R[100]mm/sec CNT100;
   1:  PR[GP1:91,1] = PR[GP1:90,1] + -19.149;
   1:  PR[GP1:91,2] = PR[GP1:90,2] + 30.505;
   1:L PR[91] R[100]mm/sec CNT100;
   1:  PR[GP1:91,1] = PR[GP1:90,1] + -27.841;
   1:  PR[GP1:91,2] = PR[GP1:90,2] + 33.809;
   1:L PR[91] R[100]mm/sec CNT100;
   1:  PR[GP1:91,1] = PR[GP1:90,1] + -31.403;
   1:  PR[GP1:91,2] = PR[GP1:90,2] + 34.332;
   1:L PR[91] R[100]mm/sec CNT100;
   1:  PR[GP1:91,1] = PR[GP1:90,1] + -38.152;
   1:  PR[GP1:91,2] = PR[GP1:90,2] + 34.812;
   1:L PR[91] R[100]mm/sec CNT100;
   1:  PR[GP1:91,1] = PR[GP1:90,1] + -44.262;
   1:  PR[GP1:91,2] = PR[GP1:90,2] + 33.827;
   1:L PR[91] R[100]mm/sec CNT100;
   1:  PR[GP1:91,1] = PR[GP1:90,1] + -48.565;
   1:  PR[GP1:91,2] = PR[GP1:90,2] + 32.864;
   1:L PR[91] R[100]mm/sec CNT100;
   1:  PR[GP1:91,1] = PR[GP1:90,1] + -55.953;
   1:  PR[GP1:91,2] = PR[GP1:90,2] + 29.148;
   1:L PR[91] R[100]mm/sec CNT100;
   1:  PR[GP1:91,1] = PR[GP1:90,1] + -58.120;
   1:  PR[GP1:91,2] = PR[GP1:90,2] + 27.927;
   1:L PR[91] R[100]mm/sec CNT100;
   1:  PR[GP1:91,1] = PR[GP1:90,1] + -65.051;
   1:  PR[GP1:91,2] = PR[GP1:90,2] + 21.127;
   1:L PR[91] R[100]mm/sec CNT100;
   1:  PR[GP1:91,1] = PR[GP1:90,1] + -65.829;
   1:  PR[GP1:91,2] = PR[GP1:90,2] + 20.307;
   1:L PR[91] R[100]mm/sec CNT100;
   1:  PR[GP1:91,1] = PR[GP1:90,1] + -70.843;
   1:  PR[GP1:91,2] = PR[GP1:90,2] + 10.658;
   1:L PR[91] R[100]mm/sec CNT100;
   1:  PR[GP1:91,1] = PR[GP1:90,1] + -72.588;
   1:  PR[GP1:91,2] = PR[GP1:90,2] + -0.072;
   1:L PR[91] R[100]mm/sec CNT100;
   1:  PR[GP1:91,1] = PR[GP1:90,1] + -70.842;
   1:  PR[GP1:91,2] = PR[GP1:90,2] + -10.808;
   1:L PR[91] R[100]mm/sec CNT100;
   1:  PR[GP1:91,1] = PR[GP1:90,1] + -70.686;
   1:  PR[GP1:91,2] = PR[GP1:90,2] + -11.124;
   1:L PR[91] R[100]mm/sec CNT100;
   1:  PR[GP1:91,1] = PR[GP1:90,1] + -65.830;
   1:  PR[GP1:91,2] = PR[GP1:90,2] + -20.450;
   1:L PR[91] R[100]mm/sec CNT100;
   1:  PR[GP1:91,1] = PR[GP1:90,1] + -65.051;
   1:  PR[GP1:91,2] = PR[GP1:90,2] + -21.271;
   1:L PR[91] R[100]mm/sec CNT100;
   1:  PR[GP1:91,1] = PR[GP1:90,1] + -58.120;
   1:  PR[GP1:91,2] = PR[GP1:90,2] + -28.071;
   1:L PR[91] R[100]mm/sec CNT100;
   1:  PR[GP1:91,1] = PR[GP1:90,1] + -55.953;
   1:  PR[GP1:91,2] = PR[GP1:90,2] + -29.292;
   1:L PR[91] R[100]mm/sec CNT100;
   1:  PR[GP1:91,1] = PR[GP1:90,1] + -48.565;
   1:  PR[GP1:91,2] = PR[GP1:90,2] + -33.008;
   1:L PR[91] R[100]mm/sec CNT100;
   1:  PR[GP1:91,1] = PR[GP1:90,1] + -44.262;
   1:  PR[GP1:91,2] = PR[GP1:90,2] + -33.971;
   1:L PR[91] R[100]mm/sec CNT100;
   1:  PR[GP1:91,1] = PR[GP1:90,1] + -38.152;
   1:  PR[GP1:91,2] = PR[GP1:90,2] + -34.956;
   1:L PR[91] R[100]mm/sec CNT100;
   1:  PR[GP1:91,1] = PR[GP1:90,1] + -31.403;
   1:  PR[GP1:91,2] = PR[GP1:90,2] + -34.476;
   1:L PR[91] R[100]mm/sec CNT100;
   1:  PR[GP1:91,1] = PR[GP1:90,1] + -27.841;
   1:  PR[GP1:91,2] = PR[GP1:90,2] + -33.953;
   1:L PR[91] R[100]mm/sec CNT100;
   1:  PR[GP1:91,1] = PR[GP1:90,1] + -19.149;
   1:  PR[GP1:91,2] = PR[GP1:90,2] + -30.649;
   1:L PR[91] R[100]mm/sec CNT100;
   1:  PR[GP1:91,1] = PR[GP1:90,1] + -18.434;
   1:  PR[GP1:91,2] = PR[GP1:90,2] + -30.300;
   1:L PR[91] R[100]mm/sec CNT100;
   1:  PR[GP1:91,1] = PR[GP1:90,1] + -15.687;
   1:  PR[GP1:91,2] = PR[GP1:90,2] + -28.180;
   1:L PR[91] R[100]mm/sec CNT100;
   1:  PR[GP1:91,1] = PR[GP1:90,1] + -10.651;
   1:  PR[GP1:91,2] = PR[GP1:90,2] + -24.491;
   1:L PR[91] R[100]mm/sec CNT100;
   1:  PR[GP1:91,1] = PR[GP1:90,1] + -10.051;
   1:  PR[GP1:91,2] = PR[GP1:90,2] + -24.013;
   1:L PR[91] R[100]mm/sec CNT100;
   1:  PR[GP1:91,1] = PR[GP1:90,1] + -9.357;
   1:  PR[GP1:91,2] = PR[GP1:90,2] + -23.202;
   1:L PR[91] R[100]mm/sec CNT100;
   1:  PR[GP1:91,1] = PR[GP1:90,1] + -4.450;
   1:  PR[GP1:91,2] = PR[GP1:90,2] + -16.491;
   1:L PR[91] R[100]mm/sec CNT100;
   1:  PR[GP1:91,1] = PR[GP1:90,1] + -3.025;
   1:  PR[GP1:91,2] = PR[GP1:90,2] + -14.891;
   1:L PR[91] R[100]mm/sec CNT100;
   1:  PR[GP1:91,1] = PR[GP1:90,1] + -1.098;
   1:  PR[GP1:91,2] = PR[GP1:90,2] + -13.764;
   1:L PR[91] R[100]mm/sec CNT100;
   1:  PR[GP1:91,1] = PR[GP1:90,1] + 1.385;
   1:  PR[GP1:91,2] = PR[GP1:90,2] + -13.740;
   1:L PR[91] R[100]mm/sec CNT100;
   1:  PR[GP1:91,1] = PR[GP1:90,1] + 2.672;
   1:  PR[GP1:91,2] = PR[GP1:90,2] + -15.282;
   1:L PR[91] R[100]mm/sec CNT100;
   1:  PR[GP1:91,1] = PR[GP1:90,1] + 3.394;
   1:  PR[GP1:91,2] = PR[GP1:90,2] + -15.737;
   1:L PR[91] R[100]mm/sec CNT100;
   1:  PR[GP1:91,1] = PR[GP1:90,1] + 4.603;
   1:  PR[GP1:91,2] = PR[GP1:90,2] + -16.399;
   1:L PR[91] R[100]mm/sec CNT100;
   1:  PR[GP1:91,1] = PR[GP1:90,1] + 9.574;
   1:  PR[GP1:91,2] = PR[GP1:90,2] + -23.199;
   1:L PR[91] R[100]mm/sec CNT100;
   1:  PR[GP1:91,1] = PR[GP1:90,1] + 10.265;
   1:  PR[GP1:91,2] = PR[GP1:90,2] + -24.009;
   1:L PR[91] R[100]mm/sec CNT100;
   1:  PR[GP1:91,1] = PR[GP1:90,1] + 15.901;
   1:  PR[GP1:91,2] = PR[GP1:90,2] + -28.182;
   1:L PR[91] R[100]mm/sec CNT100;
   1:  PR[GP1:91,1] = PR[GP1:90,1] + 18.646;
   1:  PR[GP1:91,2] = PR[GP1:90,2] + -30.303;
   1:L PR[91] R[100]mm/sec CNT100;
   1:  PR[GP1:91,1] = PR[GP1:90,1] + 19.361;
   1:  PR[GP1:91,2] = PR[GP1:90,2] + -30.652;
   1:L PR[91] R[100]mm/sec CNT100;
   1:  PR[GP1:91,1] = PR[GP1:90,1] + 28.051;
   1:  PR[GP1:91,2] = PR[GP1:90,2] + -33.951;
   1:L PR[91] R[100]mm/sec CNT100;
   1:  PR[GP1:91,1] = PR[GP1:90,1] + 31.612;
   1:  PR[GP1:91,2] = PR[GP1:90,2] + -34.475;
   1:L PR[91] R[100]mm/sec CNT100;
   1:  PR[GP1:91,1] = PR[GP1:90,1] + 38.360;
   1:  PR[GP1:91,2] = PR[GP1:90,2] + -34.956;
   1:L PR[91] R[100]mm/sec CNT100;
   1:  PR[GP1:91,1] = PR[GP1:90,1] + 44.470;
   1:  PR[GP1:91,2] = PR[GP1:90,2] + -33.972;
   1:L PR[91] R[100]mm/sec CNT100;
   1:  PR[GP1:91,1] = PR[GP1:90,1] + 48.772;
   1:  PR[GP1:91,2] = PR[GP1:90,2] + -33.007;
   1:L PR[91] R[100]mm/sec CNT100;
   1:  PR[GP1:91,1] = PR[GP1:90,1] + 56.161;
   1:  PR[GP1:91,2] = PR[GP1:90,2] + -29.297;
   1:L PR[91] R[100]mm/sec CNT100;
   1:  PR[GP1:91,1] = PR[GP1:90,1] + 58.328;
   1:  PR[GP1:91,2] = PR[GP1:90,2] + -28.078;
   1:L PR[91] R[100]mm/sec CNT100;
   1:  PR[GP1:91,1] = PR[GP1:90,1] + 65.261;
   1:  PR[GP1:91,2] = PR[GP1:90,2] + -21.267;
   1:L PR[91] R[100]mm/sec CNT100;
   1:  PR[GP1:91,1] = PR[GP1:90,1] + 66.040;
   1:  PR[GP1:91,2] = PR[GP1:90,2] + -20.444;
   1:L PR[91] R[100]mm/sec CNT100;
   1:  PR[GP1:91,1] = PR[GP1:90,1] + 71.055;
   1:  PR[GP1:91,2] = PR[GP1:90,2] + -10.820;
   1:L PR[91] R[100]mm/sec CNT100;
   1:  PR[GP1:91,1] = PR[GP1:90,1] + 72.801;
   1:  PR[GP1:91,2] = PR[GP1:90,2] + -0.072;
   1:L PR[91] R[100]mm/sec CNT100;
   1:  PR[GP1:91,1] = PR[GP1:90,1] + 71.055;
   1:  PR[GP1:91,2] = PR[GP1:90,2] + 10.676;
   1:L PR[91] R[100]mm/sec CNT100;
   1:  PR[GP1:91,1] = PR[GP1:90,1] + 66.040;
   1:  PR[GP1:91,2] = PR[GP1:90,2] + 20.300;
   1:L PR[91] R[100]mm/sec CNT100;
   1:  PR[GP1:91,1] = PR[GP1:90,1] + 65.261;
   1:  PR[GP1:91,2] = PR[GP1:90,2] + 21.123;
   1:L PR[91] R[100]mm/sec CNT100;
   1:  PR[GP1:91,1] = PR[GP1:90,1] + 58.328;
   1:  PR[GP1:91,2] = PR[GP1:90,2] + 27.934;
   1:L PR[91] R[100]mm/sec CNT100;
   1:  PR[GP1:91,1] = PR[GP1:90,1] + 56.161;
   1:  PR[GP1:91,2] = PR[GP1:90,2] + 29.153;
   1:L PR[91] R[100]mm/sec CNT100;
   1:  PR[GP1:91,1] = PR[GP1:90,1] + 48.772;
   1:  PR[GP1:91,2] = PR[GP1:90,2] + 32.863;
   1:L PR[91] R[100]mm/sec CNT100;
   1:  PR[GP1:91,1] = PR[GP1:90,1] + 44.470;
   1:  PR[GP1:91,2] = PR[GP1:90,2] + 33.828;
   1:L PR[91] R[100]mm/sec CNT100;
   1:  PR[GP1:91,1] = PR[GP1:90,1] + 38.360;
   1:  PR[GP1:91,2] = PR[GP1:90,2] + 34.812;
   1:L PR[91] R[100]mm/sec CNT100;
   1:  PR[GP1:91,1] = PR[GP1:90,1] + 31.613;
   1:  PR[GP1:91,2] = PR[GP1:90,2] + 34.331;
   1:L PR[91] R[100]mm/sec CNT100;
   1:  PR[GP1:91,1] = PR[GP1:90,1] + 28.051;
   1:  PR[GP1:91,2] = PR[GP1:90,2] + 33.807;
   1:L PR[91] R[100]mm/sec CNT100;
   1:  PR[GP1:91,1] = PR[GP1:90,1] + 19.361;
   1:  PR[GP1:91,2] = PR[GP1:90,2] + 30.508;
   1:L PR[91] R[100]mm/sec CNT100;
   1:  PR[GP1:91,1] = PR[GP1:90,1] + 18.646;
   1:  PR[GP1:91,2] = PR[GP1:90,2] + 30.159;
   1:L PR[91] R[100]mm/sec CNT100;
   1:  PR[GP1:91,1] = PR[GP1:90,1] + 15.900;
   1:  PR[GP1:91,2] = PR[GP1:90,2] + 28.037;
   1:L PR[91] R[100]mm/sec CNT100;
   1:  PR[GP1:91,1] = PR[GP1:90,1] + 10.866;
   1:  PR[GP1:91,2] = PR[GP1:90,2] + 24.347;
   1:L PR[91] R[100]mm/sec CNT100;
   1:  PR[GP1:91,1] = PR[GP1:90,1] + 10.272;
   1:  PR[GP1:91,2] = PR[GP1:90,2] + 23.873;
   1:L PR[91] R[100]mm/sec CNT100;
   1:  PR[GP1:91,1] = PR[GP1:90,1] + 9.574;
   1:  PR[GP1:91,2] = PR[GP1:90,2] + 23.055;
   1:L PR[91] R[100]mm/sec CNT100;
   1:  PR[GP1:91,1] = PR[GP1:90,1] + 4.663;
   1:  PR[GP1:91,2] = PR[GP1:90,2] + 16.338;
   1:L PR[91] R[100]mm/sec CNT100;
   1:  PR[GP1:91,1] = PR[GP1:90,1] + 3.197;
   1:  PR[GP1:91,2] = PR[GP1:90,2] + 14.724;
   1:L PR[91] R[100]mm/sec CNT100;
   1:  PR[GP1:91,1] = PR[GP1:90,1] + 1.266;
   1:  PR[GP1:91,2] = PR[GP1:90,2] + 13.597;
   1:L PR[91] R[100]mm/sec CNT100;
   1:  PR[GP1:91,1] = PR[GP1:90,1] + -1.097;
   1:  PR[GP1:91,2] = PR[GP1:90,2] + 13.620;
   1:L PR[91] R[100]mm/sec CNT100;
   1:  ! -- Layer/Ebene 53 -- !;
   1:  PR[91] = PR[90];
   1:  PR[GP1:91,1] = PR[GP1:90,1] + -3.142;
   1:  PR[GP1:91,2] = PR[GP1:90,2] + 15.299;
   1:  PR[GP1:91,3] = PR[GP1:90,3] + 32.635;
   1:L PR[91] R[100]mm/sec CNT100;
   1:  PR[GP1:91,1] = PR[GP1:90,1] + -4.515;
   1:  PR[GP1:91,2] = PR[GP1:90,2] + 16.780;
   1:L PR[91] R[100]mm/sec CNT100;
   1:  PR[GP1:91,1] = PR[GP1:90,1] + -4.526;
   1:  PR[GP1:91,2] = PR[GP1:90,2] + 16.876;
   1:L PR[91] R[100]mm/sec CNT100;
   1:  PR[GP1:91,1] = PR[GP1:90,1] + -8.744;
   1:  PR[GP1:91,2] = PR[GP1:90,2] + 22.644;
   1:L PR[91] R[100]mm/sec CNT100;
   1:  PR[GP1:91,1] = PR[GP1:90,1] + -9.849;
   1:  PR[GP1:91,2] = PR[GP1:90,2] + 23.937;
   1:L PR[91] R[100]mm/sec CNT100;
   1:  PR[GP1:91,1] = PR[GP1:90,1] + -18.453;
   1:  PR[GP1:91,2] = PR[GP1:90,2] + 30.303;
   1:L PR[91] R[100]mm/sec CNT100;
   1:  PR[GP1:91,1] = PR[GP1:90,1] + -27.906;
   1:  PR[GP1:91,2] = PR[GP1:90,2] + 33.897;
   1:L PR[91] R[100]mm/sec CNT100;
   1:  PR[GP1:91,1] = PR[GP1:90,1] + -30.604;
   1:  PR[GP1:91,2] = PR[GP1:90,2] + 34.292;
   1:L PR[91] R[100]mm/sec CNT100;
   1:  PR[GP1:91,1] = PR[GP1:90,1] + -38.186;
   1:  PR[GP1:91,2] = PR[GP1:90,2] + 34.831;
   1:L PR[91] R[100]mm/sec CNT100;
   1:  PR[GP1:91,1] = PR[GP1:90,1] + -43.494;
   1:  PR[GP1:91,2] = PR[GP1:90,2] + 33.976;
   1:L PR[91] R[100]mm/sec CNT100;
   1:  PR[GP1:91,1] = PR[GP1:90,1] + -48.557;
   1:  PR[GP1:91,2] = PR[GP1:90,2] + 32.842;
   1:L PR[91] R[100]mm/sec CNT100;
   1:  PR[GP1:91,1] = PR[GP1:90,1] + -55.275;
   1:  PR[GP1:91,2] = PR[GP1:90,2] + 29.464;
   1:L PR[91] R[100]mm/sec CNT100;
   1:  PR[GP1:91,1] = PR[GP1:90,1] + -58.070;
   1:  PR[GP1:91,2] = PR[GP1:90,2] + 27.888;
   1:L PR[91] R[100]mm/sec CNT100;
   1:  PR[GP1:91,1] = PR[GP1:90,1] + -64.508;
   1:  PR[GP1:91,2] = PR[GP1:90,2] + 21.572;
   1:L PR[91] R[100]mm/sec CNT100;
   1:  PR[GP1:91,1] = PR[GP1:90,1] + -65.744;
   1:  PR[GP1:91,2] = PR[GP1:90,2] + 20.269;
   1:L PR[91] R[100]mm/sec CNT100;
   1:  PR[GP1:91,1] = PR[GP1:90,1] + -70.305;
   1:  PR[GP1:91,2] = PR[GP1:90,2] + 11.510;
   1:L PR[91] R[100]mm/sec CNT100;
   1:  PR[GP1:91,1] = PR[GP1:90,1] + -70.733;
   1:  PR[GP1:91,2] = PR[GP1:90,2] + 10.643;
   1:L PR[91] R[100]mm/sec CNT100;
   1:  PR[GP1:91,1] = PR[GP1:90,1] + -72.371;
   1:  PR[GP1:91,2] = PR[GP1:90,2] + 0.546;
   1:L PR[91] R[100]mm/sec CNT100;
   1:  PR[GP1:91,1] = PR[GP1:90,1] + -72.494;
   1:  PR[GP1:91,2] = PR[GP1:90,2] + -0.081;
   1:L PR[91] R[100]mm/sec CNT100;
   1:  PR[GP1:91,1] = PR[GP1:90,1] + -70.860;
   1:  PR[GP1:91,2] = PR[GP1:90,2] + -9.955;
   1:L PR[91] R[100]mm/sec CNT100;
   1:  PR[GP1:91,1] = PR[GP1:90,1] + -70.732;
   1:  PR[GP1:91,2] = PR[GP1:90,2] + -10.790;
   1:L PR[91] R[100]mm/sec CNT100;
   1:  PR[GP1:91,1] = PR[GP1:90,1] + -70.305;
   1:  PR[GP1:91,2] = PR[GP1:90,2] + -11.655;
   1:L PR[91] R[100]mm/sec CNT100;
   1:  PR[GP1:91,1] = PR[GP1:90,1] + -65.744;
   1:  PR[GP1:91,2] = PR[GP1:90,2] + -20.413;
   1:L PR[91] R[100]mm/sec CNT100;
   1:  PR[GP1:91,1] = PR[GP1:90,1] + -64.508;
   1:  PR[GP1:91,2] = PR[GP1:90,2] + -21.716;
   1:L PR[91] R[100]mm/sec CNT100;
   1:  PR[GP1:91,1] = PR[GP1:90,1] + -58.070;
   1:  PR[GP1:91,2] = PR[GP1:90,2] + -28.032;
   1:L PR[91] R[100]mm/sec CNT100;
   1:  PR[GP1:91,1] = PR[GP1:90,1] + -55.275;
   1:  PR[GP1:91,2] = PR[GP1:90,2] + -29.608;
   1:L PR[91] R[100]mm/sec CNT100;
   1:  PR[GP1:91,1] = PR[GP1:90,1] + -48.557;
   1:  PR[GP1:91,2] = PR[GP1:90,2] + -32.986;
   1:L PR[91] R[100]mm/sec CNT100;
   1:  PR[GP1:91,1] = PR[GP1:90,1] + -43.494;
   1:  PR[GP1:91,2] = PR[GP1:90,2] + -34.120;
   1:L PR[91] R[100]mm/sec CNT100;
   1:  PR[GP1:91,1] = PR[GP1:90,1] + -38.186;
   1:  PR[GP1:91,2] = PR[GP1:90,2] + -34.975;
   1:L PR[91] R[100]mm/sec CNT100;
   1:  PR[GP1:91,1] = PR[GP1:90,1] + -30.604;
   1:  PR[GP1:91,2] = PR[GP1:90,2] + -34.436;
   1:L PR[91] R[100]mm/sec CNT100;
   1:  PR[GP1:91,1] = PR[GP1:90,1] + -27.906;
   1:  PR[GP1:91,2] = PR[GP1:90,2] + -34.041;
   1:L PR[91] R[100]mm/sec CNT100;
   1:  PR[GP1:91,1] = PR[GP1:90,1] + -18.474;
   1:  PR[GP1:91,2] = PR[GP1:90,2] + -30.459;
   1:L PR[91] R[100]mm/sec CNT100;
   1:  PR[GP1:91,1] = PR[GP1:90,1] + -10.823;
   1:  PR[GP1:91,2] = PR[GP1:90,2] + -24.860;
   1:L PR[91] R[100]mm/sec CNT100;
   1:  PR[GP1:91,1] = PR[GP1:90,1] + -9.856;
   1:  PR[GP1:91,2] = PR[GP1:90,2] + -24.089;
   1:L PR[91] R[100]mm/sec CNT100;
   1:  PR[GP1:91,1] = PR[GP1:90,1] + -8.744;
   1:  PR[GP1:91,2] = PR[GP1:90,2] + -22.788;
   1:L PR[91] R[100]mm/sec CNT100;
   1:  PR[GP1:91,1] = PR[GP1:90,1] + -4.414;
   1:  PR[GP1:91,2] = PR[GP1:90,2] + -16.867;
   1:L PR[91] R[100]mm/sec CNT100;
   1:  PR[GP1:91,1] = PR[GP1:90,1] + -3.147;
   1:  PR[GP1:91,2] = PR[GP1:90,2] + -15.446;
   1:L PR[91] R[100]mm/sec CNT100;
   1:  PR[GP1:91,1] = PR[GP1:90,1] + -0.994;
   1:  PR[GP1:91,2] = PR[GP1:90,2] + -14.186;
   1:L PR[91] R[100]mm/sec CNT100;
   1:  PR[GP1:91,1] = PR[GP1:90,1] + 1.287;
   1:  PR[GP1:91,2] = PR[GP1:90,2] + -14.164;
   1:L PR[91] R[100]mm/sec CNT100;
   1:  PR[GP1:91,1] = PR[GP1:90,1] + 2.458;
   1:  PR[GP1:91,2] = PR[GP1:90,2] + -15.567;
   1:L PR[91] R[100]mm/sec CNT100;
   1:  PR[GP1:91,1] = PR[GP1:90,1] + 3.099;
   1:  PR[GP1:91,2] = PR[GP1:90,2] + -15.971;
   1:L PR[91] R[100]mm/sec CNT100;
   1:  PR[GP1:91,1] = PR[GP1:90,1] + 4.569;
   1:  PR[GP1:91,2] = PR[GP1:90,2] + -16.776;
   1:L PR[91] R[100]mm/sec CNT100;
   1:  PR[GP1:91,1] = PR[GP1:90,1] + 8.962;
   1:  PR[GP1:91,2] = PR[GP1:90,2] + -22.787;
   1:L PR[91] R[100]mm/sec CNT100;
   1:  PR[GP1:91,1] = PR[GP1:90,1] + 10.074;
   1:  PR[GP1:91,2] = PR[GP1:90,2] + -24.090;
   1:L PR[91] R[100]mm/sec CNT100;
   1:  PR[GP1:91,1] = PR[GP1:90,1] + 18.666;
   1:  PR[GP1:91,2] = PR[GP1:90,2] + -30.450;
   1:L PR[91] R[100]mm/sec CNT100;
   1:  PR[GP1:91,1] = PR[GP1:90,1] + 28.117;
   1:  PR[GP1:91,2] = PR[GP1:90,2] + -34.038;
   1:L PR[91] R[100]mm/sec CNT100;
   1:  PR[GP1:91,1] = PR[GP1:90,1] + 30.814;
   1:  PR[GP1:91,2] = PR[GP1:90,2] + -34.435;
   1:L PR[91] R[100]mm/sec CNT100;
   1:  PR[GP1:91,1] = PR[GP1:90,1] + 38.395;
   1:  PR[GP1:91,2] = PR[GP1:90,2] + -34.976;
   1:L PR[91] R[100]mm/sec CNT100;
   1:  PR[GP1:91,1] = PR[GP1:90,1] + 43.702;
   1:  PR[GP1:91,2] = PR[GP1:90,2] + -34.121;
   1:L PR[91] R[100]mm/sec CNT100;
   1:  PR[GP1:91,1] = PR[GP1:90,1] + 48.765;
   1:  PR[GP1:91,2] = PR[GP1:90,2] + -32.985;
   1:L PR[91] R[100]mm/sec CNT100;
   1:  PR[GP1:91,1] = PR[GP1:90,1] + 55.484;
   1:  PR[GP1:91,2] = PR[GP1:90,2] + -29.612;
   1:L PR[91] R[100]mm/sec CNT100;
   1:  PR[GP1:91,1] = PR[GP1:90,1] + 58.278;
   1:  PR[GP1:91,2] = PR[GP1:90,2] + -28.039;
   1:L PR[91] R[100]mm/sec CNT100;
   1:  PR[GP1:91,1] = PR[GP1:90,1] + 64.718;
   1:  PR[GP1:91,2] = PR[GP1:90,2] + -21.713;
   1:L PR[91] R[100]mm/sec CNT100;
   1:  PR[GP1:91,1] = PR[GP1:90,1] + 65.955;
   1:  PR[GP1:91,2] = PR[GP1:90,2] + -20.406;
   1:L PR[91] R[100]mm/sec CNT100;
   1:  PR[GP1:91,1] = PR[GP1:90,1] + 70.518;
   1:  PR[GP1:91,2] = PR[GP1:90,2] + -11.668;
   1:L PR[91] R[100]mm/sec CNT100;
   1:  PR[GP1:91,1] = PR[GP1:90,1] + 70.946;
   1:  PR[GP1:91,2] = PR[GP1:90,2] + -10.806;
   1:L PR[91] R[100]mm/sec CNT100;
   1:  PR[GP1:91,1] = PR[GP1:90,1] + 72.584;
   1:  PR[GP1:91,2] = PR[GP1:90,2] + -0.693;
   1:L PR[91] R[100]mm/sec CNT100;
   1:  PR[GP1:91,1] = PR[GP1:90,1] + 72.707;
   1:  PR[GP1:91,2] = PR[GP1:90,2] + -0.063;
   1:L PR[91] R[100]mm/sec CNT100;
   1:  PR[GP1:91,1] = PR[GP1:90,1] + 71.072;
   1:  PR[GP1:91,2] = PR[GP1:90,2] + 9.828;
   1:L PR[91] R[100]mm/sec CNT100;
   1:  PR[GP1:91,1] = PR[GP1:90,1] + 70.945;
   1:  PR[GP1:91,2] = PR[GP1:90,2] + 10.665;
   1:L PR[91] R[100]mm/sec CNT100;
   1:  PR[GP1:91,1] = PR[GP1:90,1] + 70.518;
   1:  PR[GP1:91,2] = PR[GP1:90,2] + 11.524;
   1:L PR[91] R[100]mm/sec CNT100;
   1:  PR[GP1:91,1] = PR[GP1:90,1] + 65.955;
   1:  PR[GP1:91,2] = PR[GP1:90,2] + 20.262;
   1:L PR[91] R[100]mm/sec CNT100;
   1:  PR[GP1:91,1] = PR[GP1:90,1] + 64.718;
   1:  PR[GP1:91,2] = PR[GP1:90,2] + 21.569;
   1:L PR[91] R[100]mm/sec CNT100;
   1:  PR[GP1:91,1] = PR[GP1:90,1] + 58.278;
   1:  PR[GP1:91,2] = PR[GP1:90,2] + 27.895;
   1:L PR[91] R[100]mm/sec CNT100;
   1:  PR[GP1:91,1] = PR[GP1:90,1] + 55.484;
   1:  PR[GP1:91,2] = PR[GP1:90,2] + 29.468;
   1:L PR[91] R[100]mm/sec CNT100;
   1:  PR[GP1:91,1] = PR[GP1:90,1] + 48.765;
   1:  PR[GP1:91,2] = PR[GP1:90,2] + 32.841;
   1:L PR[91] R[100]mm/sec CNT100;
   1:  PR[GP1:91,1] = PR[GP1:90,1] + 43.702;
   1:  PR[GP1:91,2] = PR[GP1:90,2] + 33.977;
   1:L PR[91] R[100]mm/sec CNT100;
   1:  PR[GP1:91,1] = PR[GP1:90,1] + 38.395;
   1:  PR[GP1:91,2] = PR[GP1:90,2] + 34.832;
   1:L PR[91] R[100]mm/sec CNT100;
   1:  PR[GP1:91,1] = PR[GP1:90,1] + 30.814;
   1:  PR[GP1:91,2] = PR[GP1:90,2] + 34.291;
   1:L PR[91] R[100]mm/sec CNT100;
   1:  PR[GP1:91,1] = PR[GP1:90,1] + 28.117;
   1:  PR[GP1:91,2] = PR[GP1:90,2] + 33.894;
   1:L PR[91] R[100]mm/sec CNT100;
   1:  PR[GP1:91,1] = PR[GP1:90,1] + 18.665;
   1:  PR[GP1:91,2] = PR[GP1:90,2] + 30.306;
   1:L PR[91] R[100]mm/sec CNT100;
   1:  PR[GP1:91,1] = PR[GP1:90,1] + 11.040;
   1:  PR[GP1:91,2] = PR[GP1:90,2] + 24.717;
   1:L PR[91] R[100]mm/sec CNT100;
   1:  PR[GP1:91,1] = PR[GP1:90,1] + 10.081;
   1:  PR[GP1:91,2] = PR[GP1:90,2] + 23.954;
   1:L PR[91] R[100]mm/sec CNT100;
   1:  PR[GP1:91,1] = PR[GP1:90,1] + 8.962;
   1:  PR[GP1:91,2] = PR[GP1:90,2] + 22.643;
   1:L PR[91] R[100]mm/sec CNT100;
   1:  PR[GP1:91,1] = PR[GP1:90,1] + 4.629;
   1:  PR[GP1:91,2] = PR[GP1:90,2] + 16.715;
   1:L PR[91] R[100]mm/sec CNT100;
   1:  PR[GP1:91,1] = PR[GP1:90,1] + 3.326;
   1:  PR[GP1:91,2] = PR[GP1:90,2] + 15.280;
   1:L PR[91] R[100]mm/sec CNT100;
   1:  PR[GP1:91,1] = PR[GP1:90,1] + 1.168;
   1:  PR[GP1:91,2] = PR[GP1:90,2] + 14.021;
   1:L PR[91] R[100]mm/sec CNT100;
   1:  PR[GP1:91,1] = PR[GP1:90,1] + -0.994;
   1:  PR[GP1:91,2] = PR[GP1:90,2] + 14.042;
   1:L PR[91] R[100]mm/sec CNT100;
   1:  ! -- Layer/Ebene 54 -- !;
   1:  PR[91] = PR[90];
   1:  PR[GP1:91,1] = PR[GP1:90,1] + -3.265;
   1:  PR[GP1:91,2] = PR[GP1:90,2] + 15.853;
   1:  PR[GP1:91,3] = PR[GP1:90,3] + 33.245;
   1:L PR[91] R[100]mm/sec CNT100;
   1:  PR[GP1:91,1] = PR[GP1:90,1] + -4.480;
   1:  PR[GP1:91,2] = PR[GP1:90,2] + 17.164;
   1:L PR[91] R[100]mm/sec CNT100;
   1:  PR[GP1:91,1] = PR[GP1:90,1] + -4.490;
   1:  PR[GP1:91,2] = PR[GP1:90,2] + 17.253;
   1:L PR[91] R[100]mm/sec CNT100;
   1:  PR[GP1:91,1] = PR[GP1:90,1] + -8.131;
   1:  PR[GP1:91,2] = PR[GP1:90,2] + 22.231;
   1:L PR[91] R[100]mm/sec CNT100;
   1:  PR[GP1:91,1] = PR[GP1:90,1] + -9.654;
   1:  PR[GP1:91,2] = PR[GP1:90,2] + 24.013;
   1:L PR[91] R[100]mm/sec CNT100;
   1:  PR[GP1:91,1] = PR[GP1:90,1] + -17.361;
   1:  PR[GP1:91,2] = PR[GP1:90,2] + 29.715;
   1:L PR[91] R[100]mm/sec CNT100;
